(* PRIORITY 08 *)
nPriority := 8;
IF in.bR20_RC_Temperature			THEN
	out.nR20_RCTemperature			:= -1;
	fbTxBuffer[nPriority](
		IN							:= F_DIOC_20_MESSAGE_OUT(nRegister := DIOC_R01_REGISTER_REQUEST, nValue := RC_R20_RC_TEMPERATURE),
		RD							:= bTxBuffer_Read,			(* Not functional *)
		WD							:= in.bR20_RC_Temperature,
		fifo						:= ADR(TxBuffer[nPriority, 0]));
END_IF
IF in.bR21_Read_PS_AC_Voltage		THEN
	out.nR21_PsAcVoltageLevel		:= -1;
	fbTxBuffer[nPriority](
		IN							:= F_DIOC_20_MESSAGE_OUT(nRegister := DIOC_R01_REGISTER_REQUEST, nValue := RC_R21_PS_AC_VOLTAGE_LEVEL),
		RD							:= bTxBuffer_Read,			(* Not functional *)
		WD							:= in.bR21_Read_PS_AC_Voltage,
		fifo						:= ADR(TxBuffer[nPriority, 0]));
END_IF
IF in.bR22_Status_Dip_Switches		THEN
	out.sR22_Dipswitch				:= '';
	fbTxBuffer[nPriority](
		IN							:= F_DIOC_20_MESSAGE_OUT(nRegister := DIOC_R01_REGISTER_REQUEST, nValue := RC_R22_STATUS_BITS_DIPSWITCHES),
		RD							:= bTxBuffer_Read,			(* Not functional *)
		WD							:= in.bR22_Status_Dip_Switches,
		fifo						:= ADR(TxBuffer[nPriority, 0]));
END_IF
IF in.bR27_Heating_T				THEN
	out.nR27_HeatingTempHvacWater	:= -1;
	fbTxBuffer[nPriority](
		IN							:= F_DIOC_20_MESSAGE_OUT(nRegister := DIOC_R01_REGISTER_REQUEST, nValue := RC_R27_HEATING_12_13_TEMP_HVAC_WATER),
		RD							:= bTxBuffer_Read,			(* Not functional *)
		WD							:= in.bR27_Heating_T,
		fifo						:= ADR(TxBuffer[nPriority, 0]));
END_IF
IF in.bR34_Cooling_T				THEN
	out.nR34_CoolingTempIceWater	:= -1;
	fbTxBuffer[nPriority](
		IN							:= F_DIOC_20_MESSAGE_OUT(nRegister := DIOC_R01_REGISTER_REQUEST, nValue := RC_R34_COOLING_25_26_TEMP_ICE_WATER),
		RD							:= bTxBuffer_Read,			(* Not functional *)
		WD							:= in.bR34_Cooling_T,
		fifo						:= ADR(TxBuffer[nPriority, 0]));
END_IF
IF in.bR40_Pulsion_FB				THEN
	out.nR40_Pulsion_FB				:= -1;
	fbTxBuffer[nPriority](
		IN							:= F_DIOC_20_MESSAGE_OUT(nRegister := DIOC_R01_REGISTER_REQUEST, nValue := RC_R40_PULSION_17_POSITION_FEEDBACK),
		RD							:= bTxBuffer_Read,			(* Not functional *)
		WD							:= in.bR40_Pulsion_FB,
		fifo						:= ADR(TxBuffer[nPriority, 0]));
END_IF
IF in.bR42_Pulsion_T				THEN
	out.nR42_PulsionAirTemperature	:= -1;
	fbTxBuffer[nPriority](
		IN							:= F_DIOC_20_MESSAGE_OUT(nRegister := DIOC_R01_REGISTER_REQUEST, nValue := RC_R42_PULSION_18_AIR_TEMPERATURE),
		RD							:= bTxBuffer_Read,			(* Not functional *)
		WD							:= in.bR42_Pulsion_T,
		fifo						:= ADR(TxBuffer[nPriority, 0]));
END_IF
IF in.bR46_Extraction_FB			THEN
	out.nR46_Extraction_FB			:= -1;
	fbTxBuffer[nPriority](
		IN							:= F_DIOC_20_MESSAGE_OUT(nRegister := DIOC_R01_REGISTER_REQUEST, nValue := RC_R46_EXTRACTION_30_POSITION_FEEDBACK),
		RD							:= bTxBuffer_Read,			(* Not functional *)
		WD							:= in.bR46_Extraction_FB,
		fifo						:= ADR(TxBuffer[nPriority, 0]));
END_IF
IF in.bR49_Extraction_T				THEN
	out.nR49_ExtractionAirTemperature	:= -1;
	fbTxBuffer[nPriority](
		IN							:= F_DIOC_20_MESSAGE_OUT(nRegister := DIOC_R01_REGISTER_REQUEST, nValue := RC_R49_EXTRACTION_31_AIR_TEMPERATURE),
		RD							:= bTxBuffer_Read,			(* Not functional *)
		WD							:= in.bR49_Extraction_T,
		fifo						:= ADR(TxBuffer[nPriority, 0]));
END_IF
END_ACTION

ACTION Startup:
;
END_ACTION

END_FUNCTION_BLOCK

// POUs/DIOC/RC/_Internal/FB_RC_COMM
FUNCTION_BLOCK FB_RC_COMM
VAR_INPUT
	in									: ST_RC_IN;
	iPowerCycleGroup					: INT;
END_VAR
VAR_OUTPUT
	out									: ST_RC_OUT;
	nError								: E_RC_ERROR;
END_VAR
VAR CONSTANT
	TYPE_ID								: DWORD		:= 2;		(* Device identifier *)
	DEVICE_CHARGE_TIME					: TIME 		:= T#2s;	(* Optional charge time *)
	SYNC_MESSAGE_REPEAT					: TIME 		:= T#5s;	(* Sync message repeat at startup *)
	DIOC_LENGTH							: INT 		:= 21;		(* Dioc protocol length *)
	SYNC_MESSAGE						: DWORD		:= 2#0000_0000_000_1_1010_1010_1010_1111111_0;		(* Sync request = request type id *)
	SYNC_MESSAGE_HIGH					: DWORD		:= 2#0000_0000_000_1_0101_0101_0101_0101010_0;		(* Sync request = request type id *)
END_VAR
VAR
(* TC3 attribute, will be ignored by TC2 *)
{attribute 'hide_all_locals'}
(* TC2 attribute, will be ignored by TC3 *)
{library private}
	(*Startup list *)
	bStartup							: BOOL 		:= TRUE;
	bRestarted							: BOOL;					(* Device hardware restart detected by dioc *)

	(* Buffer communication *)
	Dioc_Register_IN					: ST_DIOC_REGISTER;		(* Message retrieved from buffer *)
	bRxBuffer_Read						: BOOL;
	bRxBuffer_Write						: BOOL;

	(* Fifo Buffers *)
	RxBuffer							: ARRAY[0..DIOC_RXTX_BUFFERSIZE] OF A_DIOC_MESSAGE;	(* 1 message queue *)
	TxBuffer							: ARRAY[0..DIOC_MAXPRIORITY, 0..DIOC_RXTX_BUFFERSIZE] OF A_DIOC_MESSAGE;	(* 1 message queue / priority, HIGHEST: 0 = internal priority *)

	(* Fifo Buffer handlers *)
	fbRxBuffer							: FB_DIOC_FIFO;									(* 1 message queue *)
	fbTxBuffer							: ARRAY[0..DIOC_MAXPRIORITY] OF FB_DIOC_FIFO;	(* 1 message queue / priority *)

	(* Dioc base communication layer *)
	fbDioc								: FB_DIOC;
	(* Device general register handling *)
	fbDioc_Gen							: FB_DIOC_GEN;
	(* Device specific register handling *)
	fbDioc_RC							: FB_DIOC_RC;

	i									: INT;
END_VAR

(*
	startup *)
IF bStartup THEN Startup(); END_IF
fbDioc.iPowerCycleGroup := iPowerCycleGroup;
(*
	Buffer status feedback, must be set BEFORE fb calls 
bRxBufferFull				:= fbDioc.bRxBufferFull;
bRxBufferEmpty				:= fbDioc.bRxBufferEmpty;
bTxBufferFull				:= fbDioc.bTxBufferFull;
bTxBufferEmpty				:= fbDioc.bTxBufferEmpty;*)

(*
	Get next message from message queue *)
bRxBuffer_Read				:= NOT fbDioc.out.bRxBufferEmpty;
fbRxBuffer(
	RD						:= bRxBuffer_Read,
	WD						:= bRxBuffer_Write,				(* Not functional *)
	fifo					:= ADR(RxBuffer));
Dioc_Register_IN := F_DIOC_20_MESSAGE_IN(fbRxBuffer.OUT);

(* Device Dioc base register handling and startup parameter loading *)
fbDioc_Gen(
	in						:= in.DIOC_Gen,
	in_Dioc_Status			:= fbDioc.Out,
	TYPE_ID					:= TYPE_ID,
	Dioc_Register_IN		:= Dioc_Register_IN,
	RxBuffer				:= RxBuffer,
	TxBuffer				:= TxBuffer,
	fbRxBuffer				:= fbRxBuffer,
	fbTxBuffer				:= fbTxBuffer,
	arrstStartupParameter	:= in.DIOC_RC.arrstStartupParameter,
	bRestarted				:= bRestarted,
	out						=> out.DIOC_Gen,
	nError					=>
	);
in.DIOC_Gen 				:= fbDioc_Gen.in;				(* Copy possibly changed inputs back to upper level *)

(* Device specific register handling *)
fbDioc_RC(
	in						:= in.DIOC_RC,
	in_Dioc_Status			:= fbDioc.Out,
	in_Dioc_Gen_Status		:= fbDioc_Gen.Out,
	Dioc_Register_IN		:= Dioc_Register_IN,
	RxBuffer				:= RxBuffer,
	TxBuffer				:= TxBuffer,
	fbRxBuffer				:= fbRxBuffer,
	fbTxBuffer				:= fbTxBuffer,
	bRestarted				:= bRestarted,
	out						=> out.DIOC_RC,
	nError					=>
	);
in.DIOC_RC					:= fbDioc_RC.in;				(* Copy possibly changed inputs back to upper level *)

(*
	Dioc communication layer *)
fbDioc.in.bEnable			:= in.bEnable;	(* Debug *)
fbDioc(
	DEVICE_CHARGE_TIME		:= DEVICE_CHARGE_TIME,
	DIOC_LENGTH				:= DIOC_LENGTH,
	RxBuffer				:= RxBuffer,
	TxBuffer				:= TxBuffer,
	fbRxBuffer				:= fbRxBuffer,
	fbTxBuffer				:= fbTxBuffer,
	Out						=>
	);

(*
	First loop finished *)
bStartup 					:= FALSE;

ACTION Startup:
(*
	Startup parameters *) 

(* Reset parameters
FOR i := 1 TO DIOC_NOOFSTARTUPPARAMETERS DO
	arrstStartupParameter[i].nRegister		:= 255;	(* Set to invalid *)
	arrstStartupParameter[i].nValue			:= 0;
END_FOR*)

(* Test Set parameters, switch relays
arrstStartupParameter[1].nRegister			:= 25;
arrstStartupParameter[1].nValue				:= 3;
arrstStartupParameter[2].nRegister			:= 32;
arrstStartupParameter[2].nValue				:= 3;
arrstStartupParameter[3].nRegister			:= 52;
arrstStartupParameter[3].nValue				:= 1;
arrstStartupParameter[4].nRegister			:= 25;
arrstStartupParameter[4].nValue				:= 1;
arrstStartupParameter[5].nRegister			:= 32;
arrstStartupParameter[5].nValue				:= 1;
arrstStartupParameter[6].nRegister			:= 52;
arrstStartupParameter[6].nValue				:= 2;
arrstStartupParameter[7].nRegister			:= 25;
arrstStartupParameter[7].nValue				:= 0;
arrstStartupParameter[8].nRegister			:= 32;
arrstStartupParameter[8].nValue				:= 0;
arrstStartupParameter[9].nRegister			:= 52;
arrstStartupParameter[9].nValue				:= 0;  *)


;
END_ACTION

END_FUNCTION_BLOCK

// POUs/DIOC/RC/FB_RC
FUNCTION_BLOCK FB_RC
VAR_INPUT

(*Enable bit*)
	bEn:BOOL:=TRUE; (*enable bit*)

(*input booleans*)
	bEnableFan : BOOL; (*enable fan bit (relay pin 41-42)*)

	bHeating_3P_plus :BOOL; (*Heating plus signal (output pin 7)*)
	bHeating_3P_min :BOOL; (*Heating min signal (output pin 8)*)

	bCooling_3P_plus :BOOL; (*Cooling plus signal (output pin 20)*)
	bCooling_3P_min :BOOL; (*Cooling min signal (output pin 21)*)

	bFireDamper_OPN: BOOL; (*open signal fire damper (output pin 33)*)
	bFireDamper_CLS: BOOL; (*close signal fire damper (output pin 34)*)

	bRelais_45 :BOOL; (*relay pin 45 (DO3)*)
	bRelais_46 :BOOL; (*relay pin 46 (DO2)*)
	bRelais_47 :BOOL; (*relay pin 47 (DO1)*)

(* retrieval times of all sensors*)
	iIntervalACVoltage: UDINT := 19; (*retrieval time ac voltage (in seconds)*)
	iIntervalTempHeatingWater: UDINT := 11; (*retrieval time temperature heating water (in seconds)*)
	iIntervalTempICEWater: UDINT := 9; (*retrieval time temperature ice water (in seconds)*)
	iInterval_FB_Pulsion: UDINT := 7; (*retrieval time feedback pulsion (in seconds)*)
	iIntervalTempAirPulsion: UDINT := 13; (*retrieval time temperature pulsion air (in seconds)*)
	iInterval_FB_Extraction: UDINT := 17; (*retrieval time feedback extraction (in seconds)*)
	iIntervalTempAirExtraction: UDINT := 19; (*retrieval time temperature extraction (in seconds)*)
	iIntervalDipswitches: UDINT := 17; (*retrieval time dipswitches (in seconds)*)
	iIntervalFBFiredamper: UDINT := 19; (*retrieval time feedback firedamper (in seconds)*)
	iIntervalFanFaultStatus: UDINT := 23; (*retrieval time fan fault (in seconds)*)

(* interval send times of Setpoints *)
	iSendIntervalSpHeating: INT  := 9; (*send interval time for the heating set point in seconds*)
	iSendIntervalSpCooling: INT  := 11; (*send interval time for the cooling set point in seconds*)
	iSendIntervalSpPulsion: INT  := 12; (*send interval time for the pulsion set point in seconds*)
	iSendIntervalSpExtraction: INT  := 13; (*send interval time for the extraction set point in seconds*)
	iSendIntervalSpFan: INT  := 15; (*send interval time for the fan set point in seconds*)

(* Force send setpoints *)
	bForceSendSpHeating 	: BOOL := FALSE; (*Set this to true to send the heating set point immediatly*)
	bForceSendSpCooling 	: BOOL := FALSE; (*Set this to true to send the cooling set point immediatly*)
	bForceSendSpPulsion 	: BOOL := FALSE; (*Set this to true to send the pulsion set point immediatly*)
	bForceSendSpExtraction 	: BOOL := FALSE; (*Set this to true to send the extraction set point immediatly*)
	bForceSendSpFan 		: BOOL := FALSE; (*Set this to true to send the fan set point immediatly*)

(* RC setpoints*)
	iSpHeating : INT; (*heating setpoint in %*)
	iSpCooling : INT; (*cooling setpoint in %*)
	iSpPulsion : INT; (*pulsion setpoint in %*)
	iSpExtraction : INT; (*extraction setpoint in %*)
	iSpFan : INT; (*fan setpoint in %*)

(* bool for the reset of the RC*)
	bReset:BOOL := TRUE; (*if true: resets the Room Controller*)

END_VAR
VAR_INPUT PERSISTENT

(* comment for every connection is visible on the VISU*)
	arr_sConnectionComments	: ARRAY [1..41] OF STRING(8) :=[
		'comment','comment','comment','comment','comment','comment','comment','comment','comment','comment',
		'comment','comment','comment','comment','comment','comment','comment','comment','comment','comment',
		'comment','comment','comment','comment','comment','comment','comment','comment','comment','comment',
		'comment','comment','comment','comment','comment','comment','comment','comment','comment','comment',
		'comment']; (*comments for every connection that is visible on the visualisation*)

END_VAR
VAR_OUTPUT
(*FireDamper Feedback*)
	qbFiredamperFB_OPN : BOOL; (*feedback firedamper open (input pin 37)*)
	qbFiredamperFB_CLS : BOOL; (*feedback firedamper closed (input pin 36)*)
	qbFanFault : BOOL; (*fan fault (input pin 43)*)

(* dipswitches*)
	qarr_bDipSwitches : ARRAY[1..12] OF BOOL; (*status dipswitches*)

(*measurements *)
	qfACVoltageLevel: REAL; (*measured ac voltage*)
	qfTempHeatingWater : REAL; (*temperature heating water in °C (PT1000 pin 12-13)*)
	qfTempIceWater : REAL; (*temperature ice water in °C (PT 1000 pin 25-26)*)
	qfPulsionFB : REAL; (*pulsion vav feedback in % (pin 17)*)
	qfTempAirPulsion : REAL; (*temperature pulsion in °C (PT1000 pin 18-19)*)
	qfExtractionFB : REAL; (*extraction vav feedback in % (pin 30)*)
	qfTempAirExtraction : REAL; (*temperature extraction in °C (PT1000 pin 31-32)*)

(*Analyse data*)
	qdtVersionHw: DATE;(*Hardware version of the dioc device*)
	qdtVersionSw: DATE;(*software version of the dioc device*)
	qdtVersionReg: DATE;(*register version of the dioc device*)
	qsUniqueId: STRING;(*Unique id the dioc device*)
	qrVoltageLevelA: REAL;(*Voltage level on the DIOC-A line*)
	qrVoltageLevelB: REAL;(*Voltage level on the DIOC-B line*)
	qbDeviceActive: BOOL;(*True if the device is active*)
END_VAR
VAR
(* TC3 attribute, will be ignored by TC2 *)
{attribute 'hide_all_locals'}
(* TC2 attribute, will be ignored by TC3 *)
{library private}

(*Force setpoint triggers*)
	_RtrigForceSendSpHeating: R_TRIG;
	_RtrigForceSendSpCooling: R_TRIG;
	_RtrigForceSendSpPulsion: R_TRIG;
	_RtrigForceSendSpExtraction: R_TRIG;
	_RtrigForceSendSpFan: R_TRIG;

(*SP Send Timers*)
	_tonSendIntervalSpHeating: TON;
	_tonSendIntervalSpCooling: TON;
	_tonSendIntervalSpPulsion: TON;
	_tonSendIntervalSpExtraction: TON;
	_tonSendIntervalSpFan: TON;

(* reset variabelen *)
	_iReset_Counter:INT;

(* startup variabelen *)
	_RtrigCalibration:R_TRIG;
	_FtrigCalibration:F_TRIG;
	_iLostCalibration:INT;
	_iStateInit:INT;
	_iStateInit_Counter:INT;
	_iStartupListNumber: INT := 1;
	_bFirstCycle: BOOL := TRUE;
	_iLoadbalance : INT;

(* visualisatie variabelen*)
	_iVis: INT;
	_bSelected : BOOL;
	_bAnalyse	:BOOL;
	_bPrevVisu : BOOL;
	_bNextVisu :BOOL;
	_RtrigAnalyse :R_TRIG;
	_RtrigSim :R_TRIG;
	_bSim : BOOL;
	_bComments : BOOL;

	_iSpHeatingSim : INT;
	_iSpCoolingSim : INT;
	_iSpPulsionSim : INT;
	_iSpExtractionSim : INT;
	_iSpFanSim : INT;

	_bEnableFanSim : BOOL;
	_bHeating_3P_plusSim :BOOL;
	_bHeating_3P_minSim :BOOL;
	_bCooling_3P_plusSim :BOOL;
	_bCooling_3P_minSim :BOOL;
	_bFireDamper_OPNSim: BOOL;
	_bFireDamper_CLSSim: BOOL;
	_bRelais_45Sim : BOOL;
	_bRelais_46Sim : BOOL;
	_bRelais_47Sim : BOOL;

(*start*)
	_bInit : BOOL := FALSE;

(*functionblock for communication with RC *)
	FB_DIOC_COMM : FB_RC_COMM;

END_VAR

(*Wait 0.5s to start the next DIOC device, charging too many DIOC devices at once will give too much current*)
IF NOT _bInit THEN
    DIOC_tonLastStart(IN:=TRUE , PT:= T#500ms);
    IF  NOT DIOC_tonLastStart.Q THEN
    	RETURN;
    END_IF
    DIOC_tonLastStart(IN:=FALSE , PT:= T#500ms); (*resets the timer*)
    _bInit := TRUE;
END_IF

(* falling and rising edge RC calibration*)
_RtrigCalibration(CLK:= FB_DIOC_COMM.out.DIOC_Gen.bDeviceActive, Q=> );
_FtrigCalibration(CLK:= FB_DIOC_COMM.out.DIOC_Gen.bDeviceActive, Q=> );

(* enable reset the device when calibration is lost for 30 cycles. *)
IF _FtrigCalibration.Q THEN
	_iLostCalibration := 1;
END_IF

IF _iLostCalibration = 30 THEN
	bReset := TRUE;
END_IF

IF _iLostCalibration < 30 AND _iLostCalibration > 0 AND NOT FB_DIOC_COMM.out.DIOC_Gen.bDeviceActive THEN
	_iLostCalibration := _iLostCalibration + 1;
ELSE
	_iLostCalibration := 0;
END_IF

(* reset the device when breset is high, cut off power to device for 1000 cycles to make sure the device has lost all power*)
IF breset OR DIOC_bRestart OR NOT bEn THEN
	_iReset_Counter := 0;
	FB_DIOC_COMM.in.bEnable := FALSE;
	breset := FALSE;
END_IF

IF _iReset_Counter < 1000 THEN
	IF _iReset_Counter = 999 THEN
	    _bInit := FALSE;
	END_IF
	_iReset_Counter := _iReset_Counter +1;
	_iStateInit := 0;
ELSE
	FB_DIOC_COMM.in.bEnable := bEn;
END_IF

(* send startuplist, send all values that need to be sent at startup + set automatic response types of certain measurements,
with synchronisations added in between the messages to not disrupt the flow of the startparameters *)

IF _bFirstCycle THEN
	StartupList();
END_IF

(* request all static info when the device has been active for some time *)
stateinit();

_RtrigSim(CLK:= _bSim, Q=> );
IF _RtrigSim.q THEN
	(* limit analog values from 0% to 100% *)
	iSpHeating := LIMIT(0,iSpHeating,100);
	iSpCooling := LIMIT(0,iSpCooling,100);
	iSpPulsion := LIMIT(0,iSpPulsion,100);
	iSpExtraction := LIMIT(0,iSpExtraction,100);
	iSpFan := LIMIT(0,iSpFan,100);

	_iSpHeatingSim  := iSpHeating;
	_iSpCoolingSim  := iSpCooling;
	_iSpPulsionSim  := iSpPulsion;
	_iSpExtractionSim  := iSpExtraction;
	_iSpFanSim  := iSpFan;

	_bEnableFanSim := bEnableFan;
	_bHeating_3P_plusSim := bHeating_3P_plus;
	_bHeating_3P_minSim := bHeating_3P_min;
	_bCooling_3P_plusSim := bCooling_3P_plus;
	_bCooling_3P_minSim := bCooling_3P_min;
	_bFireDamper_OPNSim:= bFireDamper_OPN;
	_bFireDamper_CLSSim:= bFireDamper_CLS;
END_IF

(*Forward setpoints*)
_RtrigForceSendSpHeating(CLK:= bForceSendSpHeating);
bForceSendSpHeating := FALSE;
_tonSendIntervalSpHeating(IN:= NOT _tonSendIntervalSpHeating.q, PT:= UDINT_TO_TIME(INT_TO_UDINT(iSendIntervalSpHeating * 1000)));
IF _tonSendIntervalSpHeating.Q OR _RtrigForceSendSpHeating.Q THEN
	(* limit analog values from 0% to 100% *)
	iSpHeating := LIMIT(0,iSpHeating,100);
	FB_DIOC_COMM.in.DIOC_RC.nR26_Heating_SP := INT_TO_UINT(TRUNC_INT(INT_TO_REAL( SEL(_bSim, iSpHeating, _iSpHeatingSim)) / 100* 4090));
	FB_DIOC_COMM.in.DIOC_RC.bR26_Heating_SP := TRUE;
END_IF;

_RtrigForceSendSpCooling(CLK:= bForceSendSpCooling);
bForceSendSpCooling := FALSE;
_tonSendIntervalSpCooling(IN:= NOT _tonSendIntervalSpCooling.q, PT:= UDINT_TO_TIME(INT_TO_UDINT(iSendIntervalSpCooling * 1000)));
IF _tonSendIntervalSpCooling.Q OR _RtrigForceSendSpCooling.Q  THEN
	(* limit analog values from 0% to 100% *)
	iSpCooling := LIMIT(0,iSpCooling,100);
	FB_DIOC_COMM.in.DIOC_RC.nR33_Cooling_SP := INT_TO_UINT(TRUNC_INT(INT_TO_REAL( SEL(_bSim, iSpCooling, _iSpCoolingSim)) / 100* 4090));
	FB_DIOC_COMM.in.DIOC_RC.bR33_Cooling_SP := TRUE;
END_IF;

_RtrigForceSendSpPulsion(CLK:= bForceSendSpPulsion);
bForceSendSpPulsion := FALSE;
_tonSendIntervalSpPulsion(IN:= NOT _tonSendIntervalSpPulsion.q, PT:= UDINT_TO_TIME(INT_TO_UDINT(iSendIntervalSpPulsion * 1000)));
IF _tonSendIntervalSpPulsion.Q OR _RtrigForceSendSpPulsion.Q   THEN
	(* limit analog values from 0% to 100% *)
	iSpPulsion := LIMIT(0,iSpPulsion,100);
	FB_DIOC_COMM.in.DIOC_RC.nR39_Pulsion_SP := INT_TO_UINT(TRUNC_INT(INT_TO_REAL( SEL(_bSim, iSpPulsion, _iSpPulsionSim)) / 100* 4090));
	FB_DIOC_COMM.in.DIOC_RC.bR39_Pulsion_SP := TRUE;
END_IF;

_RtrigForceSendSpExtraction(CLK:= bForceSendSpExtraction);
bForceSendSpExtraction := FALSE;
_tonSendIntervalSpExtraction(IN:= NOT _tonSendIntervalSpExtraction.q, PT:= UDINT_TO_TIME(INT_TO_UDINT(iSendIntervalSpExtraction * 1000)));
IF _tonSendIntervalSpExtraction.Q OR _RtrigForceSendSpExtraction.Q   THEN
	(* limit analog values from 0% to 100% *)
	iSpExtraction := LIMIT(0,iSpExtraction,100);
	FB_DIOC_COMM.in.DIOC_RC.nR45_Extraction_SP := INT_TO_UINT(TRUNC_INT(INT_TO_REAL( SEL(_bSim, iSpExtraction, _iSpExtractionSim)) / 100* 4090));
	FB_DIOC_COMM.in.DIOC_RC.bR45_Extraction_SP := TRUE;
END_IF;

_RtrigForceSendSpFan(CLK:= bForceSendSpFan);
bForceSendSpFan := FALSE;
_tonSendIntervalSpFan(IN:= NOT _tonSendIntervalSpFan.q, PT:= UDINT_TO_TIME(INT_TO_UDINT(iSendIntervalSpFan * 1000)));
IF _tonSendIntervalSpFan.Q  OR _RtrigForceSendSpFan.Q  THEN
	(* limit analog values from 0% to 100% *)
	iSpFan := LIMIT(0,iSpFan,100);
	FB_DIOC_COMM.in.DIOC_RC.nR56_Fan_SP := INT_TO_UINT(TRUNC_INT(INT_TO_REAL( SEL(_bSim, iSpFan, _iSpFanSim)) /100* 4090));
	FB_DIOC_COMM.in.DIOC_RC.bR56_Fan_SP := TRUE;
END_IF;

(* call communication block *)
FB_DIOC_COMM(in:= , out=> , nError=> );

(*Inputs*)
qarr_bDipSwitches[1] := FB_DIOC_COMM.out.DIOC_RC.bR22_Dipswitch_S01;
qarr_bDipSwitches[2] := FB_DIOC_COMM.out.DIOC_RC.bR22_Dipswitch_S02;
qarr_bDipSwitches[3] := FB_DIOC_COMM.out.DIOC_RC.bR22_Dipswitch_S03;
qarr_bDipSwitches[4] := FB_DIOC_COMM.out.DIOC_RC.bR22_Dipswitch_S04;
qarr_bDipSwitches[5] := FB_DIOC_COMM.out.DIOC_RC.bR22_Dipswitch_S05;
qarr_bDipSwitches[6] := FB_DIOC_COMM.out.DIOC_RC.bR22_Dipswitch_S06;
qarr_bDipSwitches[7] := FB_DIOC_COMM.out.DIOC_RC.bR22_Dipswitch_S07;
qarr_bDipSwitches[8] := FB_DIOC_COMM.out.DIOC_RC.bR22_Dipswitch_S08;
qarr_bDipSwitches[9] := FB_DIOC_COMM.out.DIOC_RC.bR22_Dipswitch_S09;
qarr_bDipSwitches[10] := FB_DIOC_COMM.out.DIOC_RC.bR22_Dipswitch_S10;
qarr_bDipSwitches[11] := FB_DIOC_COMM.out.DIOC_RC.bR22_Dipswitch_S11;
qarr_bDipSwitches[12] := FB_DIOC_COMM.out.DIOC_RC.bR22_Dipswitch_S12;

qbFiredamperFB_OPN := FB_DIOC_COMM.out.DIOC_RC.bR53_FireDamperFB_OPN;
qbFiredamperFB_CLS := FB_DIOC_COMM.out.DIOC_RC.bR53_FireDamperFB_CLS;
qbFanFault := FB_DIOC_COMM.out.DIOC_RC.bR58_FanFaultStatus;

(*Measurements *)
qfACVoltageLevel:=FB_DIOC_COMM.out.DIOC_RC.nR21_PsAcVoltageLevel;
qfTempHeatingWater:=FB_DIOC_COMM.out.DIOC_RC.nR27_HeatingTempHvacWater;
qfTempIceWater:=FB_DIOC_COMM.out.DIOC_RC.nR34_CoolingTempIceWater;
qfPulsionFB:=FB_DIOC_COMM.out.DIOC_RC.nR40_Pulsion_FB;
qfTempAirPulsion:=FB_DIOC_COMM.out.DIOC_RC.nR42_PulsionAirTemperature;
qfExtractionFB:=FB_DIOC_COMM.out.DIOC_RC.nR46_Extraction_FB;
qfTempAirExtraction:=FB_DIOC_COMM.out.DIOC_RC.nR49_ExtractionAirTemperature;

(*Outputs*)
FB_DIOC_COMM.in.DIOC_RC.bR25_Heating_7_8_3p_min := SEL(_bSim, bHeating_3P_min, _bHeating_3P_minSim);
FB_DIOC_COMM.in.DIOC_RC.bR25_Heating_7_8_3p_plus_pwm := SEL(_bSim, bHeating_3P_plus, _bHeating_3P_plusSim);

FB_DIOC_COMM.in.DIOC_RC.bR32_Cooling_20_21_3p_min := SEL(_bSim, bCooling_3P_min, _bCooling_3P_minSim);
FB_DIOC_COMM.in.DIOC_RC.bR32_Cooling_20_21_3p_plus_pwm := SEL(_bSim, bCooling_3P_plus, _bCooling_3P_plusSim);

FB_DIOC_COMM.in.DIOC_RC.bR52_FireDamperCOM_NC := SEL(_bSim, bFireDamper_CLS, _bFireDamper_CLSSim);
FB_DIOC_COMM.in.DIOC_RC.bR52_FireDamperCOM_NO := SEL(_bSim, bFireDamper_OPN, _bFireDamper_OPNSim);

FB_DIOC_COMM.in.DIOC_RC.bR57_Fan_Enable := SEL(_bSim, bEnableFan, _bEnableFanSim);

FB_DIOC_COMM.in.DIOC_RC.bR61_do_45 := SEL(_bSim, bRelais_45, _bRelais_45Sim);
FB_DIOC_COMM.in.DIOC_RC.bR61_do_46 := SEL(_bSim, bRelais_46, _bRelais_46Sim);
FB_DIOC_COMM.in.DIOC_RC.bR61_do_47 := SEL(_bSim, bRelais_47, _bRelais_47Sim);


(*loadbalance, only do these tasks every 47 cycles to save time *)
_iLoadbalance := _iLoadbalance + 1;
IF _iLoadbalance > 47 THEN
	_iLoadbalance := 0;

	(*save static info*)
	qdtVersionHw:=FB_DIOC_COMM.out.DIOC_Gen.dtR04_VersionHW;
	qdtVersionSw:=FB_DIOC_COMM.out.DIOC_Gen.dtR05_VersionSW;
	qdtVersionReg:=FB_DIOC_COMM.out.DIOC_Gen.dtR06_VersionREG;
	qsUniqueId:=FB_DIOC_COMM.out.DIOC_Gen.sR07_UniqueID;
	
	qrVoltageLevelA:=FB_DIOC_COMM.out.DIOC_Gen.nR09_DiocVoltageA;
	qrVoltageLevelB:=FB_DIOC_COMM.out.DIOC_Gen.nR10_DiocVoltageB;

	qbDeviceActive:=FB_DIOC_COMM.out.DIOC_Gen.bDeviceActive;
END_IF;

(* Visualisation *)
(*
_RtrigAnalyse(CLK:= _bAnalyse, Q=> );
IF _RtrigAnalyse.q  AND (CurrentVisu <> DIOC_DEBUGSCHERM) AND DIOC_Debug THEN
	DIOC_DebugLinkPrevScreen:=CurrentVisu;
	CurrentVisu := DIOC_DEBUGSCHERM;
END_IF
IF _bAnalyse AND DIOC_Debug THEN
	DIOC_pDebugged_RC := ADRINST();
	_bAnalyse := FALSE;
END_IF*)

IF _bSelected = FALSE THEN
	_bSim := FALSE;
	_iVis := 0;
END_IF;

IF _bNextVisu THEN
	_iVis := _iVis + 1;
	_bNextVisu := FALSE;
END_IF

IF _bPrevVisu THEN
	_iVis := _iVis - 1;
	_bPrevVisu := FALSE;
END_IF

IF _iVis > 0 THEN
	_iVis := 0;
END_IF;

IF _iVis < 0 THEN
	_iVis := 0;
END_IF;

_bFirstCycle := FALSE;

ACTION StartupList:
_iStartupListNumber := 1;
(*change transmit offset*)
FB_DIOC_COMM.in.DIOC_RC.arrstStartupParameter[_iStartupListNumber].nRegister:=DIOC_R84_TRANSMIT_DELAY;
FB_DIOC_COMM.in.DIOC_RC.arrstStartupParameter[_iStartupListNumber].nValue:=30;

_iStartupListNumber := _iStartupListNumber +1;
FB_DIOC_COMM.in.DIOC_RC.arrstStartupParameter[_iStartupListNumber].nRegister:=DIOC_R02_REGISTER_INTERVAL;
FB_DIOC_COMM.in.DIOC_RC.arrstStartupParameter[_iStartupListNumber].nValue:=19;

_iStartupListNumber := _iStartupListNumber +1;
FB_DIOC_COMM.in.DIOC_RC.arrstStartupParameter[_iStartupListNumber].nRegister:=DIOC_R01_REGISTER_REQUEST;
FB_DIOC_COMM.in.DIOC_RC.arrstStartupParameter[_iStartupListNumber].nValue:=INT_TO_DWORD(DIOC_R84_TRANSMIT_DELAY);

(*device enabled*)
FB_DIOC_COMM.in.DIOC_RC.arrstStartupParameter[_iStartupListNumber].nRegister:=DIOC_R02_REGISTER_INTERVAL;
FB_DIOC_COMM.in.DIOC_RC.arrstStartupParameter[_iStartupListNumber].nValue:=15;

_iStartupListNumber := _iStartupListNumber +1;
FB_DIOC_COMM.in.DIOC_RC.arrstStartupParameter[_iStartupListNumber].nRegister:=DIOC_R01_REGISTER_REQUEST;
FB_DIOC_COMM.in.DIOC_RC.arrstStartupParameter[_iStartupListNumber].nValue:=INT_TO_DWORD(DIOC_R11_DEVICE_ENABLE);

(*voltage level A*)
_iStartupListNumber := _iStartupListNumber +1;
FB_DIOC_COMM.in.DIOC_RC.arrstStartupParameter[_iStartupListNumber].nRegister:=DIOC_R02_REGISTER_INTERVAL;
FB_DIOC_COMM.in.DIOC_RC.arrstStartupParameter[_iStartupListNumber].nValue:=59;

_iStartupListNumber := _iStartupListNumber +1;
FB_DIOC_COMM.in.DIOC_RC.arrstStartupParameter[_iStartupListNumber].nRegister:=DIOC_R01_REGISTER_REQUEST;
FB_DIOC_COMM.in.DIOC_RC.arrstStartupParameter[_iStartupListNumber].nValue:=INT_TO_DWORD(DIOC_R09_VOLTAGE_LEVEL_A);

(*voltage level B*)
_iStartupListNumber := _iStartupListNumber +1;
FB_DIOC_COMM.in.DIOC_RC.arrstStartupParameter[_iStartupListNumber].nRegister:=DIOC_R02_REGISTER_INTERVAL;
FB_DIOC_COMM.in.DIOC_RC.arrstStartupParameter[_iStartupListNumber].nValue:=61;

_iStartupListNumber := _iStartupListNumber +1;
FB_DIOC_COMM.in.DIOC_RC.arrstStartupParameter[_iStartupListNumber].nRegister:=DIOC_R01_REGISTER_REQUEST;
FB_DIOC_COMM.in.DIOC_RC.arrstStartupParameter[_iStartupListNumber].nValue:=INT_TO_DWORD(DIOC_R10_VOLTAGE_LEVEL_B);

(*AC PS Voltage level*)
_iStartupListNumber := _iStartupListNumber +1;
FB_DIOC_COMM.in.DIOC_RC.arrstStartupParameter[_iStartupListNumber].nRegister:=DIOC_R02_REGISTER_INTERVAL;
FB_DIOC_COMM.in.DIOC_RC.arrstStartupParameter[_iStartupListNumber].nValue:=iIntervalACVoltage;

_iStartupListNumber := _iStartupListNumber +1;
FB_DIOC_COMM.in.DIOC_RC.arrstStartupParameter[_iStartupListNumber].nRegister:=DIOC_R01_REGISTER_REQUEST;
FB_DIOC_COMM.in.DIOC_RC.arrstStartupParameter[_iStartupListNumber].nValue:=INT_TO_DWORD(RC_R21_PS_AC_VOLTAGE_LEVEL);

(* Heating 12-13 temperature HVAC water *)
_iStartupListNumber := _iStartupListNumber +1;
FB_DIOC_COMM.in.DIOC_RC.arrstStartupParameter[_iStartupListNumber].nRegister:=DIOC_R02_REGISTER_INTERVAL;
FB_DIOC_COMM.in.DIOC_RC.arrstStartupParameter[_iStartupListNumber].nValue:=iIntervalTempHeatingWater;

_iStartupListNumber := _iStartupListNumber +1;
FB_DIOC_COMM.in.DIOC_RC.arrstStartupParameter[_iStartupListNumber].nRegister:=DIOC_R01_REGISTER_REQUEST;
FB_DIOC_COMM.in.DIOC_RC.arrstStartupParameter[_iStartupListNumber].nValue:= INT_TO_DWORD(RC_R27_HEATING_12_13_TEMP_HVAC_WATER);

(*sync*)
_iStartupListNumber := _iStartupListNumber +1;
FB_DIOC_COMM.in.DIOC_RC.arrstStartupParameter[_iStartupListNumber].nRegister:=85;
FB_DIOC_COMM.in.DIOC_RC.arrstStartupParameter[_iStartupListNumber].nValue:=2730;

(*Cooling 25-26 temperature ICE water *)
_iStartupListNumber := _iStartupListNumber +1;
FB_DIOC_COMM.in.DIOC_RC.arrstStartupParameter[_iStartupListNumber].nRegister:=DIOC_R02_REGISTER_INTERVAL;
FB_DIOC_COMM.in.DIOC_RC.arrstStartupParameter[_iStartupListNumber].nValue:=iIntervalTempICEWater;

_iStartupListNumber := _iStartupListNumber +1;
FB_DIOC_COMM.in.DIOC_RC.arrstStartupParameter[_iStartupListNumber].nRegister:=DIOC_R01_REGISTER_REQUEST;
FB_DIOC_COMM.in.DIOC_RC.arrstStartupParameter[_iStartupListNumber].nValue:=INT_TO_DWORD(RC_R34_COOLING_25_26_TEMP_ICE_WATER);

(* Pulsion_FB *)
_iStartupListNumber := _iStartupListNumber +1;
FB_DIOC_COMM.in.DIOC_RC.arrstStartupParameter[_iStartupListNumber].nRegister:=DIOC_R02_REGISTER_INTERVAL;
FB_DIOC_COMM.in.DIOC_RC.arrstStartupParameter[_iStartupListNumber].nValue:=iInterval_FB_Pulsion;

_iStartupListNumber := _iStartupListNumber +1;
FB_DIOC_COMM.in.DIOC_RC.arrstStartupParameter[_iStartupListNumber].nRegister:=DIOC_R01_REGISTER_REQUEST;
FB_DIOC_COMM.in.DIOC_RC.arrstStartupParameter[_iStartupListNumber].nValue:=INT_TO_DWORD(RC_R40_PULSION_17_POSITION_FEEDBACK);

(* Pulsion Air Temperature *)
_iStartupListNumber := _iStartupListNumber +1;
FB_DIOC_COMM.in.DIOC_RC.arrstStartupParameter[_iStartupListNumber].nRegister:=DIOC_R02_REGISTER_INTERVAL;
FB_DIOC_COMM.in.DIOC_RC.arrstStartupParameter[_iStartupListNumber].nValue:=iIntervalTempAirPulsion;

_iStartupListNumber := _iStartupListNumber +1;
FB_DIOC_COMM.in.DIOC_RC.arrstStartupParameter[_iStartupListNumber].nRegister:=DIOC_R01_REGISTER_REQUEST;
FB_DIOC_COMM.in.DIOC_RC.arrstStartupParameter[_iStartupListNumber].nValue:=INT_TO_DWORD(RC_R42_PULSION_18_AIR_TEMPERATURE);

(*sync*)
_iStartupListNumber := _iStartupListNumber +1;
FB_DIOC_COMM.in.DIOC_RC.arrstStartupParameter[_iStartupListNumber].nRegister:=85;
FB_DIOC_COMM.in.DIOC_RC.arrstStartupParameter[_iStartupListNumber].nValue:=2730;

(* Extraction_FB *)
_iStartupListNumber := _iStartupListNumber +1;
FB_DIOC_COMM.in.DIOC_RC.arrstStartupParameter[_iStartupListNumber].nRegister:=DIOC_R02_REGISTER_INTERVAL;
FB_DIOC_COMM.in.DIOC_RC.arrstStartupParameter[_iStartupListNumber].nValue:=iInterval_FB_Extraction;

_iStartupListNumber := _iStartupListNumber +1;
FB_DIOC_COMM.in.DIOC_RC.arrstStartupParameter[_iStartupListNumber].nRegister:=DIOC_R01_REGISTER_REQUEST;
FB_DIOC_COMM.in.DIOC_RC.arrstStartupParameter[_iStartupListNumber].nValue:=INT_TO_DWORD(RC_R46_EXTRACTION_30_POSITION_FEEDBACK);

(* Extraction Air Temperature *)
_iStartupListNumber := _iStartupListNumber +1;
FB_DIOC_COMM.in.DIOC_RC.arrstStartupParameter[_iStartupListNumber].nRegister:=DIOC_R02_REGISTER_INTERVAL;
FB_DIOC_COMM.in.DIOC_RC.arrstStartupParameter[_iStartupListNumber].nValue:=iIntervalTempAirExtraction;

_iStartupListNumber := _iStartupListNumber +1;
FB_DIOC_COMM.in.DIOC_RC.arrstStartupParameter[_iStartupListNumber].nRegister:=DIOC_R01_REGISTER_REQUEST;
FB_DIOC_COMM.in.DIOC_RC.arrstStartupParameter[_iStartupListNumber].nValue:=INT_TO_DWORD(RC_R49_EXTRACTION_31_AIR_TEMPERATURE);

(* Dipswitches *)
_iStartupListNumber := _iStartupListNumber +1;
FB_DIOC_COMM.in.DIOC_RC.arrstStartupParameter[_iStartupListNumber].nRegister:=DIOC_R02_REGISTER_INTERVAL;
FB_DIOC_COMM.in.DIOC_RC.arrstStartupParameter[_iStartupListNumber].nValue:=iIntervalDipswitches;

_iStartupListNumber := _iStartupListNumber +1;
FB_DIOC_COMM.in.DIOC_RC.arrstStartupParameter[_iStartupListNumber].nRegister:=DIOC_R01_REGISTER_REQUEST;
FB_DIOC_COMM.in.DIOC_RC.arrstStartupParameter[_iStartupListNumber].nValue:=INT_TO_DWORD(RC_R22_STATUS_BITS_DIPSWITCHES);

(* FB_Firedamper *)
_iStartupListNumber := _iStartupListNumber +1;
FB_DIOC_COMM.in.DIOC_RC.arrstStartupParameter[_iStartupListNumber].nRegister:=DIOC_R02_REGISTER_INTERVAL;
FB_DIOC_COMM.in.DIOC_RC.arrstStartupParameter[_iStartupListNumber].nValue:=iIntervalFBFiredamper;

_iStartupListNumber := _iStartupListNumber +1;
FB_DIOC_COMM.in.DIOC_RC.arrstStartupParameter[_iStartupListNumber].nRegister:=DIOC_R01_REGISTER_REQUEST;
FB_DIOC_COMM.in.DIOC_RC.arrstStartupParameter[_iStartupListNumber].nValue:=INT_TO_DWORD(RC_R53_FIREDAMPER_36_37_FEEDBACK);

(* fan fault status *)
_iStartupListNumber := _iStartupListNumber +1;
FB_DIOC_COMM.in.DIOC_RC.arrstStartupParameter[_iStartupListNumber].nRegister:=DIOC_R02_REGISTER_INTERVAL;
FB_DIOC_COMM.in.DIOC_RC.arrstStartupParameter[_iStartupListNumber].nValue:=iIntervalFanFaultStatus;

_iStartupListNumber := _iStartupListNumber +1;
FB_DIOC_COMM.in.DIOC_RC.arrstStartupParameter[_iStartupListNumber].nRegister:=DIOC_R01_REGISTER_REQUEST;
FB_DIOC_COMM.in.DIOC_RC.arrstStartupParameter[_iStartupListNumber].nValue:=INT_TO_DWORD(RC_R58_FAN_FAULT_STATUS);

(*sync*)
_iStartupListNumber := _iStartupListNumber +1;
FB_DIOC_COMM.in.DIOC_RC.arrstStartupParameter[_iStartupListNumber].nRegister:=85;
FB_DIOC_COMM.in.DIOC_RC.arrstStartupParameter[_iStartupListNumber].nValue:=2730;
END_ACTION

ACTION Stateinit:
(* Gradually request all static information at startup of the RC *)
CASE _iStateInit OF
	0:
		IF _RtrigCalibration.Q  THEN
		_iStateInit:=1;
		END_IF
	1:
		_iStateInit_Counter:=_iStateInit_Counter+1;
		IF _iStateInit_Counter>4000 THEN
			_iStateInit:=_iStateInit+1;
			_iStateInit_Counter:=0;
		END_IF
	2:
		FB_DIOC_COMM.in.DIOC_Gen.bR04_Request_HW_Version:=TRUE;
		_iStateInit:=_iStateInit+1;
	3:
		_iStateInit_Counter:=_iStateInit_Counter+1;
		IF FB_DIOC_COMM.out.DIOC_Gen.dtR04_VersionHW <> DWORD_TO_DATE(0) THEN
			_iStateInit:=_iStateInit+1;
			_iStateInit_Counter:=0;
		ELSE
			IF _iStateInit_Counter>1000 THEN
				FB_DIOC_COMM.in.DIOC_Gen.bR04_Request_HW_Version:=TRUE;
				_iStateInit_Counter:=0;
			END_IF
		END_IF
	4:
		FB_DIOC_COMM.in.DIOC_Gen.bR05_Request_SW_Version:=TRUE;
		_iStateInit:=_iStateInit+1;
	5:
			_iStateInit_Counter:=_iStateInit_Counter+1;
		IF FB_DIOC_COMM.out.DIOC_Gen.dtR05_VersionSW <> DWORD_TO_DATE(0) THEN
			_iStateInit:=_iStateInit+1;
			_iStateInit_Counter:=0;
		ELSE
			IF _iStateInit_Counter>1000 THEN
				FB_DIOC_COMM.in.DIOC_Gen.bR05_Request_SW_Version:=TRUE;
				_iStateInit_Counter:=0;
			END_IF
		END_IF
	6:
		FB_DIOC_COMM.in.DIOC_Gen.bR06_Request_Register_Version:=TRUE;
		_iStateInit:=_iStateInit+1;
	7:
			_iStateInit_Counter:=_iStateInit_Counter+1;
		IF FB_DIOC_COMM.out.DIOC_Gen.dtR06_VersionREG <> DWORD_TO_DATE(0) THEN
			_iStateInit:=_iStateInit+1;
			_iStateInit_Counter:=0;
		ELSE
			IF _iStateInit_Counter>1000 THEN
				FB_DIOC_COMM.in.DIOC_Gen.bR06_Request_Register_Version:=TRUE;
				_iStateInit_Counter:=0;
			END_IF
		END_IF
	8:
		FB_DIOC_COMM.in.DIOC_Gen.bR07_Request_Unique_ID:=TRUE;
		_iStateInit:=_iStateInit+1;
	9:
		_iStateInit_Counter:=_iStateInit_Counter+1;
		IF FB_DIOC_COMM.out.DIOC_Gen.sR07_UniqueID <> '' THEN
			_iStateInit:=_iStateInit+1;
			_iStateInit_Counter:=0;
		ELSE
			IF _iStateInit_Counter>800 THEN
				FB_DIOC_COMM.in.DIOC_Gen.bR07_Request_Unique_ID:=TRUE;
				_iStateInit_Counter:=0;
			END_IF
		END_IF
	10:
		_iStateInit := 0;
END_CASE
END_ACTION

END_FUNCTION_BLOCK

// POUs/DIOC/TP10/_Internal/FB_DIOC_TP10
FUNCTION_BLOCK FB_DIOC_TP10
VAR_INPUT
	(* Data handshake interface *)
	in									: ST_DIOC_TP10_IN;
	in_Dioc_Status						: ST_DIOC_OUT;			(* Feedback dioc communication block *)
	in_Dioc_Gen_Status					: ST_DIOC_GEN_OUT;		(* Feedback general registers *)
	(*bDeviceReady						: BOOL;					(* Device charged and ready *)
	bDeviceActive						: BOOL;					(* Device is active *)*)
	Dioc_Register_IN					: ST_DIOC_REGISTER;		(* Message retrieved from buffer *)
	(* Buffer statusses *)
	bRxBufferFull						: BOOL;
	bRxBufferEmpty						: BOOL;
	bTxBufferFull						: BOOL;
	bTxBufferEmpty						: BOOL;
END_VAR
VAR_OUTPUT
	(* RC feedback data *)
	out									: ST_DIOC_TP10_OUT;
	nError								: E_DIOC_TP10_ERROR;
	qbBufferFull						: BOOL;
END_VAR
VAR_IN_OUT
	(*Dioc_Register_OUT					: A_DIOC_MESSAGE;*)
	RxBuffer							: ARRAY[0..DIOC_RXTX_BUFFERSIZE] OF A_DIOC_MESSAGE;	(* 1 message queue *)
	TxBuffer							: ARRAY[0..DIOC_MAXPRIORITY, 0..DIOC_RXTX_BUFFERSIZE] OF A_DIOC_MESSAGE;	(* 1 message queue / priority, HIGHEST: 0 = internal priority *)
	(* Fifo Buffer handlers *)
	fbRxBuffer							: FB_DIOC_FIFO;									(* 1 message queue *)
	fbTxBuffer							: ARRAY[0..DIOC_MAXPRIORITY] OF FB_DIOC_FIFO;	(* 1 message queue / priority *)
	(* Restarted ? *)
	bRestarted							: BOOL;
END_VAR
VAR
(* TC3 attribute, will be ignored by TC2 *)
{attribute 'hide_all_locals'}
(* TC2 attribute, will be ignored by TC3 *)
{library private}
	(* Previous state in *)
	stDeviceDataInPrevious				: ST_DIOC_TP10_IN;

	(*
		Timer sync message *)
	tSync								: TON;

	(*
		dioc communication *)
	stDiocRegister						: ST_DIOC_REGISTER;
	stDiocMessage						: A_DIOC_MESSAGE;

	(*
		Sync message response, response is constructed at runtime, can depend on device *)
	dwSyncMessageResponse				: DWORD;

	(*
		device data IN, request to the device *)
	fpDeviceDataInNew					: R_TRIG;

	(*
		Startup list *)
	bStartup							: BOOL 		:= TRUE;

	iRefreshCycles						: INT;
	_FtrigCalibration					:F_TRIG;

	(* various *)
	i									: INT;
	byToggle							: BYTE;
	nPriority							: INT;		(* This value avoids copy paste errors, filled in by the program, see send action *)

	(* TEMP VARS *)
	nWriteRegister				 		: A_DIOC_DATA_TYPE;
	(* Buffer read / write *)
	bRxBuffer_Read						: BOOL;
	bRxBuffer_Write						: BOOL;
	bTxBuffer_Read						: BOOL;
	bTxBuffer_Write						: BOOL;

	(* Current values *)
	sR07_UniqueID						: STRING[24];				(* TEMP R7: Unique ID *)
	sR07_UniqueID_hex					: STRING[2];				(* TEMP R7: Unique ID *)

	nTemp: DINT;
	byParity							: BYTE; (*Byte to determine parity*)
	iNoButtonParity: INT;


	outRef									: ST_DIOC_TP10_OUT;
END_VAR

(* © 2016 FixSus BVBA all rights reserved *)
(* © Handles TP10 specific variables of the TP10 *)
(*	startup *)
IF bStartup THEN Startup(); END_IF

(*
	Toggle byte *)
byToggle		:= byToggle + 1;

(* handle restart *)
IF	bRestarted				THEN
	Restart();
END_IF

(*refresh sent data every 1000 cycles*)
IF iRefreshCycles < 1000 THEN
	iRefreshCycles := iRefreshCycles +1;
ELSIF in_Dioc_Gen_Status.nR10_DiocVoltageB > -1 THEN
	iRefreshCycles := 0;
END_IF;

(*on loss of calibration reset all values to 0*)
_FtrigCalibration(CLK:= in_Dioc_Gen_Status.bDeviceActive, Q=> );

IF _FtrigCalibration.Q THEN
	out.nR50_TouchButtonStatus			:= 0;
	out.bR50_TouchButton01				:= out.nR50_TouchButtonStatus.0;
	out.bR50_TouchButton02				:= out.nR50_TouchButtonStatus.1;
	out.bR50_TouchButton03				:= out.nR50_TouchButtonStatus.2;
	out.bR50_TouchButton04				:= out.nR50_TouchButtonStatus.3;
	out.bR50_TouchButton05				:= out.nR50_TouchButtonStatus.4;
	out.bR50_TouchButton06				:= out.nR50_TouchButtonStatus.5;
	out.bR50_TouchButton07				:= out.nR50_TouchButtonStatus.6;
	out.bR50_TouchButton08				:= out.nR50_TouchButtonStatus.7;
	out.bR50_TouchButton09				:= out.nR50_TouchButtonStatus.8;
	out.bR50_TouchButton10				:= out.nR50_TouchButtonStatus.9;
	out.nR21_RoomTemperature 			:= 0;
	out.nR27_VOC			 			:= 0;
	out.nR25_CO2			 			:= 0;
	out.nR23_ROOM_HUMIDITY	 			:= 0;
	out.nR35_ROOM_ILLUMINATION_LUXL_VALUE 	:= 0;
	out.nR36_ROOM_ILLUMINATION_LUXH_VALUE	:= 0;
	out.nR37_ROOM_ILLUMINATION_IRL_VALUE 	:= 0;
	out.nR38_ROOM_ILLUMINATION_IRH_VALUE 	:= 0;
END_IF;
(*
	Process new data from dioc *)
Receive();

(*
	External Dioc request processing, with priority handling *)
Send();

(*
	First loop finished *)
bStartup 					:= FALSE;

ACTION Receive:
(* !!! ONLY ACTIVE WHEN THE DEVICE IS ACTIVE !!! *)

(*New dioc data received and the device is active *)
IF in_Dioc_Status.bRxBufferEmpty	OR NOT in_Dioc_Gen_Status.bDeviceActive THEN
	RETURN;
END_IF

(*Process new data *)
CASE Dioc_Register_IN.nRegister			OF



	TP10_R19_CONFIGURATION_SETUP:
		out.nR19_CONFIGURATION_SETUP 		:= Dioc_Register_IN.nValue;

		out.nR19_ROOMTEMPERATURE_AVAILABLE	:= out.nR19_CONFIGURATION_SETUP.0;
		out.nR19_HUMIDITY_AVAILABLE  		:= out.nR19_CONFIGURATION_SETUP.1;
		out.nR19_CO2_AVAILABLE  			:= out.nR19_CONFIGURATION_SETUP.2;
		out.nR19_VOC_AVAILABLE  			:= out.nR19_CONFIGURATION_SETUP.3;
		out.nR19_CO_AVAILABLE  				:= out.nR19_CONFIGURATION_SETUP.4;
		out.nR19_PRESSURE_AVAILABLE  		:= out.nR19_CONFIGURATION_SETUP.5;
		out.nR19_REFPRESSURE_AVAILABLE  	:= out.nR19_CONFIGURATION_SETUP.6;
		out.nR19_ILLUMINATION_AVAILABLE  	:= out.nR19_CONFIGURATION_SETUP.7;
		out.nR19_TOUCH_AVAILABLE  			:= out.nR19_CONFIGURATION_SETUP.8;
		out.nR19_PROXIMITY_AVAILABLE  		:= out.nR19_CONFIGURATION_SETUP.9;
		out.nR19_HAPTIC_AVAILABLE  			:= out.nR19_CONFIGURATION_SETUP.10;
		out.nR19_RGB_AVAILABLE  			:= out.nR19_CONFIGURATION_SETUP.11;

	TP10_R20_ROOMTEMPERATURE_SETUP:
		out.nR20_ROOMTEMPERATURE_SETUP := DWORD_TO_REAL(Dioc_Register_IN.nValue);

	TP10_R21_ROOMTEMPERATURE: 				(* 20 *)
		out.nR21_RoomTemperature 			:= F_SCALE_FROM_DIOC(Dioc_Register_IN.nValue, 0, 4095, -20, 120, -20);

	TP10_R22_ROOM_HUMIDITY_SETUP:
		out.nR22_ROOM_HUMIDITY_SETUP := DWORD_TO_REAL(Dioc_Register_IN.nValue);


	TP10_R23_ROOM_HUMIDITY:
		out.nR23_ROOM_HUMIDITY 			:= F_SCALE_FROM_DIOC(Dioc_Register_IN.nValue, 0, 4095, 0, 100, 0);

	TP10_R24_CO2_SETUP:
		out.nR24_CO2_SETUP 	:= DWORD_TO_REAL(Dioc_Register_IN.nValue);

	TP10_R25_CO2:
		IF ( in_Dioc_Gen_Status.dtR04_VersionHW >= d#2018-06-11 ) AND ( in_Dioc_Gen_Status.dtR05_VersionSW >= d#2018-07-23 ) THEN
			(*new eCO2 sensors*)
			out.nR25_CO2		:= DWORD_TO_REAL(Dioc_Register_IN.nValue);
		ELSE
			(*old eCO2 sensors, correcton on measurement*)
			out.nR25_CO2 		:= DWORD_TO_REAL(267 + Dioc_Register_IN.nValue /3);
		END_IF

	TP10_R26_VOC_SETUP:
		out.nR26_VOC_SETUP := DWORD_TO_REAL(Dioc_Register_IN.nValue);

	TP10_R27_VOC:
		out.nR27_VOC 		:= DWORD_TO_REAL(Dioc_Register_IN.nValue);

	TP10_R28_VOC_BASELINE_L_SETUP:
			out.nR28_VOC_BASELINE_L_SETUP := Dioc_Register_IN.nValue;
			out.br29_VOC_BASELINE_VALID := TRUE;

	TP10_R29_VOC_BASELINE_H_SETUP:
			out.nR29_VOC_BASELINE_H_SETUP := Dioc_Register_IN.nValue;
			in.bR28_VOC_Baseline_L_REQ := TRUE;

	TP10_R34_ROOM_ILLUMINATION_SETUP:
		out.nR34_ROOM_ILLUMINATION_SETUP 		:= DWORD_TO_REAL(Dioc_Register_IN.nValue);

	TP10_R35_ROOM_ILLUMINATION_LUXL_VALUE:
		out.nR35_ROOM_ILLUMINATION_LUXL_VALUE 	:= SEL(Dioc_Register_IN.nValue.11,0,2) + SEL(Dioc_Register_IN.nValue.10,0,1) +SEL(Dioc_Register_IN.nValue.9,0,0.5) +SEL(Dioc_Register_IN.nValue.8,0,0.25);

	TP10_R36_ROOM_ILLUMINATION_LUXH_VALUE:
		out.nR36_ROOM_ILLUMINATION_LUXH_VALUE 	:= DWORD_TO_REAL(Dioc_Register_IN.nValue);
		in.bR35_LUX_L := TRUE;

	TP10_R37_ROOM_ILLUMINATION_IRL_VALUE:
		out.nR37_ROOM_ILLUMINATION_IRL_VALUE 	:=  SEL(Dioc_Register_IN.nValue.11,0,2) + SEL(Dioc_Register_IN.nValue.10,0,1) +SEL(Dioc_Register_IN.nValue.9,0,0.5) +SEL(Dioc_Register_IN.nValue.8,0,0.25);

	TP10_R38_ROOM_ILLUMINATION_IRH_VALUE:
		out.nR38_ROOM_ILLUMINATION_IRH_VALUE 	:= DWORD_TO_REAL(Dioc_Register_IN.nValue);
		in.bR37_IR_L := TRUE;

	TP10_R50_TOUCH_BUTTON_STATUS: (* if the received value is possible, use it, else, request it again. *)
		out.nR50_TouchButtonStatus			:= Dioc_Register_IN.nValue;
		IF 	(out.nR50_TouchButtonStatus.10 OR out.nR50_TouchButtonStatus.11) AND (iNoButtonParity > 0) THEN (* nieuwe versie met pariteit*)
			iNoButtonParity := iNoButtonParity - 1;
		END_IF;

		IF 	(NOT out.nR50_TouchButtonStatus.10) AND (NOT  out.nR50_TouchButtonStatus.11) AND (iNoButtonParity < 100) THEN (* nieuwe versie met pariteit*)
			iNoButtonParity := iNoButtonParity + 1;
		END_IF;

		IF iNoButtonParity < 10 THEN
			IF 	out.nR50_TouchButtonStatus = 2048 OR out.nR50_TouchButtonStatus = 1025 OR out.nR50_TouchButtonStatus = 1026 OR out.nR50_TouchButtonStatus = 1028 OR out.nR50_TouchButtonStatus = 1032 OR out.nR50_TouchButtonStatus = 1040 OR
		 		out.nR50_TouchButtonStatus = 1056 OR  out.nR50_TouchButtonStatus = 1088 OR out.nR50_TouchButtonStatus = 1152 OR out.nR50_TouchButtonStatus = 1280 OR out.nR50_TouchButtonStatus = 1536 THEN

				out.bR50_TouchButton01				:= out.nR50_TouchButtonStatus.0;
				out.bR50_TouchButton02				:= out.nR50_TouchButtonStatus.1;
				out.bR50_TouchButton03				:= out.nR50_TouchButtonStatus.2;
				out.bR50_TouchButton04				:= out.nR50_TouchButtonStatus.3;
				out.bR50_TouchButton05				:= out.nR50_TouchButtonStatus.4;
				out.bR50_TouchButton06				:= out.nR50_TouchButtonStatus.5;
				out.bR50_TouchButton07				:= out.nR50_TouchButtonStatus.6;
				out.bR50_TouchButton08				:= out.nR50_TouchButtonStatus.7;
				out.bR50_TouchButton09				:= out.nR50_TouchButtonStatus.8;
				out.bR50_TouchButton10				:= out.nR50_TouchButtonStatus.9;
			ELSE
				(*re-request the value*)
				in.bR50_TouchButtonStatus := TRUE;
			END_IF;

		ELSE (* versie zonder Pariteitsbits*)
			IF 	out.nR50_TouchButtonStatus = 0 OR out.nR50_TouchButtonStatus = 1 OR out.nR50_TouchButtonStatus = 2 OR out.nR50_TouchButtonStatus = 4 OR out.nR50_TouchButtonStatus = 8 OR out.nR50_TouchButtonStatus = 16 OR
		 		out.nR50_TouchButtonStatus = 32 OR  out.nR50_TouchButtonStatus = 64 OR out.nR50_TouchButtonStatus = 128 OR out.nR50_TouchButtonStatus = 256 OR out.nR50_TouchButtonStatus = 512 THEN

				out.bR50_TouchButton01				:= out.nR50_TouchButtonStatus.0;
				out.bR50_TouchButton02				:= out.nR50_TouchButtonStatus.1;
				out.bR50_TouchButton03				:= out.nR50_TouchButtonStatus.2;
				out.bR50_TouchButton04				:= out.nR50_TouchButtonStatus.3;
				out.bR50_TouchButton05				:= out.nR50_TouchButtonStatus.4;
				out.bR50_TouchButton06				:= out.nR50_TouchButtonStatus.5;
				out.bR50_TouchButton07				:= out.nR50_TouchButtonStatus.6;
				out.bR50_TouchButton08				:= out.nR50_TouchButtonStatus.7;
				out.bR50_TouchButton09				:= out.nR50_TouchButtonStatus.8;
				out.bR50_TouchButton10				:= out.nR50_TouchButtonStatus.9;
			ELSE
				(*re-request the value*)
				in.bR50_TouchButtonStatus := TRUE;
			END_IF;
		END_IF;


	TP10_R51_TOUCH_LED_STATUS:				(* 51 *)
		byParity := INT_TO_BYTE(BOOL_TO_INT(Dioc_Register_IN.nValue.0) + BOOL_TO_INT(Dioc_Register_IN.nValue.1) + BOOL_TO_INT(Dioc_Register_IN.nValue.2) + BOOL_TO_INT(Dioc_Register_IN.nValue.3) + BOOL_TO_INT(Dioc_Register_IN.nValue.4) + BOOL_TO_INT(Dioc_Register_IN.nValue.5) + BOOL_TO_INT(Dioc_Register_IN.nValue.6) + BOOL_TO_INT(Dioc_Register_IN.nValue.7) + BOOL_TO_INT(Dioc_Register_IN.nValue.8) + BOOL_TO_INT(Dioc_Register_IN.nValue.9));
		IF Dioc_Register_IN.nValue.10 = byParity.0 AND Dioc_Register_IN.nValue.11 <> byParity.0 OR (iNoButtonParity >= 10) THEN
			out.nR51_TouchLedStatus				:= Dioc_Register_IN.nValue;
		END_IF;

	TP10_R52_TOUCH_LED_MASK:				(* 52 *)
		byParity := INT_TO_BYTE(BOOL_TO_INT(Dioc_Register_IN.nValue.0) + BOOL_TO_INT(Dioc_Register_IN.nValue.1) + BOOL_TO_INT(Dioc_Register_IN.nValue.2) + BOOL_TO_INT(Dioc_Register_IN.nValue.3) + BOOL_TO_INT(Dioc_Register_IN.nValue.4) + BOOL_TO_INT(Dioc_Register_IN.nValue.5) + BOOL_TO_INT(Dioc_Register_IN.nValue.6) + BOOL_TO_INT(Dioc_Register_IN.nValue.7) + BOOL_TO_INT(Dioc_Register_IN.nValue.8) + BOOL_TO_INT(Dioc_Register_IN.nValue.9));
		IF Dioc_Register_IN.nValue.10 = byParity.0 AND Dioc_Register_IN.nValue.11 <> byParity.0 OR (iNoButtonParity >= 10) THEN
			out.nR52_TouchLedMask				:= Dioc_Register_IN.nValue;
		END_IF;

	TP10_R57_HAPTIC_INTENSITY:
		;


	ELSE;
END_CASE
END_ACTION

ACTION Restart:
(* Invalidate previous status with something impossible and not dangerous, must be something that will be updated by the cycle *)
stDeviceDataInPrevious.nR51_TouchLedStatus := 16500;
stDeviceDataInPrevious.NR83_ButtonSensitivity := 0;

out := outRef;
(* invalidate out feedback used in the send conditions *)
iRefreshCycles := 0;

(* Re-set the status of the leds *)
(*
in.nR51_TouchLedStatus		:= out.nR51_TouchLedStatus;
in.nR52_TouchLedMask		:= out.nR52_TouchLedMask;
*)

(* Acknowledge *)
bRestarted := FALSE;
END_ACTION

ACTION Send:
(* !!! ONLY ACTIVE WHEN THE DEVICE IS ACTIVE !!! *)

(*
	is the device active *)
IF NOT in_Dioc_Gen_Status.bDeviceActive THEN
	(*reset all saved values*)
	RETURN;
END_IF



(*
	New dioc data received ? *)
IF MEMCMP(ADR(stDeviceDataInPrevious), ADR(in), SIZEOF(stDeviceDataInPrevious)) = 0 THEN RETURN; END_IF;

nTemp := MEMCMP(ADR(stDeviceDataInPrevious), ADR(in), SIZEOF(stDeviceDataInPrevious));

(*opbouw RGB*)
in.nR61_RGB_MSB.0 := in.nR61_RGB_RED.4;
in.nR61_RGB_MSB.1 := in.nR61_RGB_RED.5;
in.nR61_RGB_MSB.2 := in.nR61_RGB_RED.6;
in.nR61_RGB_MSB.3 := in.nR61_RGB_RED.7;
in.nR61_RGB_MSB.4 := in.nR61_RGB_GREEN.4;
in.nR61_RGB_MSB.5 := in.nR61_RGB_GREEN.5;
in.nR61_RGB_MSB.6 := in.nR61_RGB_GREEN.6;
in.nR61_RGB_MSB.7 := in.nR61_RGB_GREEN.7;
in.nR61_RGB_MSB.8 := in.nR61_RGB_BLUE.4;
in.nR61_RGB_MSB.9 := in.nR61_RGB_BLUE.5;
in.nR61_RGB_MSB.10 := in.nR61_RGB_BLUE.6;
in.nR61_RGB_MSB.11 := in.nR61_RGB_BLUE.7;

in.nR62_RGB_LSB.0 := in.nR61_RGB_RED.0;
in.nR62_RGB_LSB.1 := in.nR61_RGB_RED.1;
in.nR62_RGB_LSB.2 := in.nR61_RGB_RED.2;
in.nR62_RGB_LSB.3 := in.nR61_RGB_RED.3;
in.nR62_RGB_LSB.4 := in.nR61_RGB_GREEN.0;
in.nR62_RGB_LSB.5 := in.nR61_RGB_GREEN.1;
in.nR62_RGB_LSB.6 := in.nR61_RGB_GREEN.2;
in.nR62_RGB_LSB.7 := in.nR61_RGB_GREEN.3;
in.nR62_RGB_LSB.8 := in.nR61_RGB_BLUE.0;
in.nR62_RGB_LSB.9 := in.nR61_RGB_BLUE.1;
in.nR62_RGB_LSB.10 := in.nR61_RGB_BLUE.2;
in.nR62_RGB_LSB.11 := in.nR61_RGB_BLUE.3;

(*
	Handle register handling in the order of priority *)
(* PRIORITY 00: internal commands (eg at startup) *)
(* Test message, highest priority, always send a sync message first *)
nPriority := 0;

(* PRIORITY 01 *)
nPriority := 1;

(* PRIORITY 02 *)
nPriority := 2;
(* PRIORITY 03 *)
nPriority := 3;
IF in.nR51_TouchLedStatus <> stDeviceDataInPrevious.nR51_TouchLedStatus  OR iRefreshCycles = 320 THEN				(* Set touch led status *)
	byParity := INT_TO_BYTE(BOOL_TO_INT(in.nR51_TouchLedStatus.0) + BOOL_TO_INT(in.nR51_TouchLedStatus.1) + BOOL_TO_INT(in.nR51_TouchLedStatus.2) + BOOL_TO_INT(in.nR51_TouchLedStatus.3) + BOOL_TO_INT(in.nR51_TouchLedStatus.4) + BOOL_TO_INT(in.nR51_TouchLedStatus.5) + BOOL_TO_INT(in.nR51_TouchLedStatus.6) + BOOL_TO_INT(in.nR51_TouchLedStatus.7) + BOOL_TO_INT(in.nR51_TouchLedStatus.8) + BOOL_TO_INT(in.nR51_TouchLedStatus.9));
	bTxBuffer_Write					:= TRUE;
	fbTxBuffer[nPriority](
		IN							:= F_DIOC_20_MESSAGE_OUT(nRegister := TP10_R51_TOUCH_LED_STATUS, nValue := SEL(byParity.0,in.nR51_TouchLedStatus+2048,in.nR51_TouchLedStatus+1024)),
		RD							:= bTxBuffer_Read,			(* Not functional *)
		WD							:= bTxBuffer_Write,
		fifo						:= ADR(TxBuffer[nPriority, 0]));
	IF NOT bTxBuffer_Write			THEN	(* Successfully transferred to the Tx Buffer *)
		stDeviceDataInPrevious.nR51_TouchLedStatus			:= in.nR51_TouchLedStatus;
	END_IF
END_IF

IF in.nR52_TouchLedMask <> stDeviceDataInPrevious.nR52_TouchLedMask  OR iRefreshCycles = 360 THEN	(* Set touch led mask *)
	byParity := INT_TO_BYTE(BOOL_TO_INT(in.nR52_TouchLedMask.0) + BOOL_TO_INT(in.nR52_TouchLedMask.1) + BOOL_TO_INT(in.nR52_TouchLedMask.2) + BOOL_TO_INT(in.nR52_TouchLedMask.3) + BOOL_TO_INT(in.nR52_TouchLedMask.4) + BOOL_TO_INT(in.nR52_TouchLedMask.5) + BOOL_TO_INT(in.nR52_TouchLedMask.6) + BOOL_TO_INT(in.nR52_TouchLedMask.7) + BOOL_TO_INT(in.nR52_TouchLedMask.8) + BOOL_TO_INT(in.nR52_TouchLedMask.9));
	bTxBuffer_Write					:= TRUE;
	fbTxBuffer[nPriority](
		IN							:= F_DIOC_20_MESSAGE_OUT(nRegister := TP10_R52_TOUCH_LED_MASK, nValue := SEL(byParity.0,in.nR52_TouchLedMask+2048,in.nR52_TouchLedMask+1024)),
		RD							:= bTxBuffer_Read,			(* Not functional *)
		WD							:= bTxBuffer_Write,
		fifo						:= ADR(TxBuffer[nPriority, 0]));
	IF NOT bTxBuffer_Write			THEN	(* Successfully transferred to the Tx Buffer *)
		stDeviceDataInPrevious.nR52_TouchLedMask			:= in.nR52_TouchLedMask;
	END_IF
END_IF
(* PRIORITY 04 *)
nPriority := 4;
IF in.NR83_ButtonSensitivity <> stDeviceDataInPrevious.NR83_ButtonSensitivity THEN	(* write the button sensitivity*)
	IF ((in.NR83_ButtonSensitivity >0) AND (in.NR83_ButtonSensitivity <100)) THEN
		bTxBuffer_Write					:= TRUE;
		fbTxBuffer[nPriority](
			IN							:= F_DIOC_20_MESSAGE_OUT(nRegister := TP10_R83_BUTTON_SENSITIVITY, nValue := in.NR83_ButtonSensitivity),
			RD							:= bTxBuffer_Read,			(* Not functional *)
			WD							:= bTxBuffer_Write,
			fifo						:= ADR(TxBuffer[nPriority, 0]));
		IF NOT bTxBuffer_Write			THEN	(* Successfully transferred to the Tx Buffer *)
			stDeviceDataInPrevious.NR83_ButtonSensitivity := in.NR83_ButtonSensitivity;
		END_IF
	END_IF
END_IF

(* PRIORITY 05 *)
nPriority := 5;

(* PRIORITY 06 *)
nPriority := 6;

(* PRIORITY 07 *)
nPriority := 7;

IF in.bR19_Configuration_Setup THEN		(* Request configuration setup*)
	fbTxBuffer[nPriority](
		IN							:= F_DIOC_20_MESSAGE_OUT(nRegister := DIOC_R01_REGISTER_REQUEST, nValue := TP10_R19_CONFIGURATION_SETUP),
		RD							:= bTxBuffer_Read,			(* Not functional *)
		WD							:= in.bR19_Configuration_Setup,
		fifo						:= ADR(TxBuffer[nPriority, 0]));
END_IF

IF in.bR20_Room_Temperature_Setup			THEN		(* Request room temperature setup*)
	bTxBuffer_Write					:= TRUE;
	fbTxBuffer[nPriority](
		IN							:= F_DIOC_20_MESSAGE_OUT(nRegister :=DIOC_R01_REGISTER_REQUEST  , nValue := TP10_R20_ROOMTEMPERATURE_SETUP),
		RD							:= bTxBuffer_Read,			(* Not functional *)
		WD							:= bTxBuffer_Write,
		fifo						:= ADR(TxBuffer[nPriority, 0]));
	in.bR20_Room_Temperature_Setup := FALSE;
END_IF

IF in.bR21_Room_Temperature			THEN		(* Request room temperature *)
	(*out.nR20_Room_Temperature		:= -1;*) (*TV // not necesairy, down point in trending software*)
	fbTxBuffer[nPriority](
		IN							:= F_DIOC_20_MESSAGE_OUT(nRegister := DIOC_R01_REGISTER_REQUEST, nValue := TP10_R21_ROOMTEMPERATURE),
		RD							:= bTxBuffer_Read,			(* Not functional *)
		WD							:= in.bR21_Room_Temperature,
		fifo						:= ADR(TxBuffer[nPriority, 0]));
END_IF

IF in.bR22_Room_Humidity_Setup			THEN		(* Request room temperature setup*)
	fbTxBuffer[nPriority](
		IN							:= F_DIOC_20_MESSAGE_OUT(nRegister :=DIOC_R01_REGISTER_REQUEST  , nValue := TP10_R22_ROOM_HUMIDITY_SETUP),
		RD							:= bTxBuffer_Read,			(* Not functional *)
		WD							:= in.bR22_Room_Humidity_Setup,
		fifo						:= ADR(TxBuffer[nPriority, 0]));
END_IF

IF in.bR24_CO2_Setup			THEN		(* Request CO2 setup*)
	fbTxBuffer[nPriority](
		IN							:= F_DIOC_20_MESSAGE_OUT(nRegister :=DIOC_R01_REGISTER_REQUEST  , nValue := TP10_R24_CO2_SETUP),
		RD							:= bTxBuffer_Read,			(* Not functional *)
		WD							:= in.bR24_CO2_Setup,
		fifo						:= ADR(TxBuffer[nPriority, 0]));
END_IF

IF in.bR26_VOC_Setup			THEN		(* Request VOC setup*)
	fbTxBuffer[nPriority](
		IN							:= F_DIOC_20_MESSAGE_OUT(nRegister :=DIOC_R01_REGISTER_REQUEST  , nValue := TP10_R26_VOC_SETUP),
		RD							:= bTxBuffer_Read,			(* Not functional *)
		WD							:= in.bR26_VOC_Setup,
		fifo						:= ADR(TxBuffer[nPriority, 0]));
END_IF

IF in.bR28_VOC_Baseline_L_REQ THEN
	fbTxBuffer[nPriority](
		IN							:= F_DIOC_20_MESSAGE_OUT(nRegister :=DIOC_R01_REGISTER_REQUEST  , nValue := TP10_R28_VOC_BASELINE_L_SETUP),
		RD							:= bTxBuffer_Read,			(* Not functional *)
		WD							:= in.bR28_VOC_Baseline_L_REQ,
		fifo						:= ADR(TxBuffer[nPriority, 0]));
END_IF;

IF in.bR28_VOC_Baseline_L_SEND THEN
	fbTxBuffer[nPriority](
		IN							:= F_DIOC_20_MESSAGE_OUT(nRegister :=TP10_R28_VOC_BASELINE_L_SETUP  , nValue := out.nR28_VOC_BASELINE_L_SETUP),
		RD							:= bTxBuffer_Read,			(* Not functional *)
		WD							:= in.bR28_VOC_Baseline_L_SEND,
		fifo						:= ADR(TxBuffer[nPriority, 0]));
END_IF;

IF in.bR29_VOC_Baseline_H_REQ THEN
	fbTxBuffer[nPriority](
		IN							:= F_DIOC_20_MESSAGE_OUT(nRegister :=DIOC_R01_REGISTER_REQUEST  , nValue := TP10_R29_VOC_BASELINE_H_SETUP),
		RD							:= bTxBuffer_Read,			(* Not functional *)
		WD							:= in.bR29_VOC_BaseLine_H_REQ,
		fifo						:= ADR(TxBuffer[nPriority, 0]));
END_IF;

IF in.bR29_VOC_Baseline_H_SEND THEN
	fbTxBuffer[nPriority](
		IN							:= F_DIOC_20_MESSAGE_OUT(nRegister :=TP10_R29_VOC_BASELINE_H_SETUP  , nValue := out.nR29_VOC_BASELINE_H_SETUP),
		RD							:= bTxBuffer_Read,			(* Not functional *)
		WD							:= in.bR29_VOC_Baseline_H_SEND,
		fifo						:= ADR(TxBuffer[nPriority, 0]));
	in.bR28_VOC_BaseLine_L_SEND := TRUE;
END_IF;

IF in.bR34_LUX_Setup THEN
	fbTxBuffer[nPriority](
		IN							:= F_DIOC_20_MESSAGE_OUT(nRegister :=DIOC_R01_REGISTER_REQUEST  , nValue := TP10_R34_ROOM_ILLUMINATION_SETUP),
		RD							:= bTxBuffer_Read,			(* Not functional *)
		WD							:= in.bR34_LUX_Setup,
		fifo						:= ADR(TxBuffer[nPriority, 0]));
END_IF

IF in.bR35_LUX_L THEN
	fbTxBuffer[nPriority](
		IN							:= F_DIOC_20_MESSAGE_OUT(nRegister :=DIOC_R01_REGISTER_REQUEST  , nValue := TP10_R35_ROOM_ILLUMINATION_LUXL_VALUE),
		RD							:= bTxBuffer_Read,			(* Not functional *)
		WD							:= in.bR35_LUX_L,
		fifo						:= ADR(TxBuffer[nPriority, 0]));
END_IF

IF in.bR36_LUX_H THEN
	fbTxBuffer[nPriority](
		IN							:= F_DIOC_20_MESSAGE_OUT(nRegister :=DIOC_R01_REGISTER_REQUEST  , nValue := TP10_R36_ROOM_ILLUMINATION_LUXH_VALUE),
		RD							:= bTxBuffer_Read,			(* Not functional *)
		WD							:= in.bR36_LUX_H,
		fifo						:= ADR(TxBuffer[nPriority, 0]));
END_IF

IF in.bR37_IR_L THEN
	fbTxBuffer[nPriority](
		IN							:= F_DIOC_20_MESSAGE_OUT(nRegister :=DIOC_R01_REGISTER_REQUEST  , nValue := TP10_R37_ROOM_ILLUMINATION_IRL_VALUE),
		RD							:= bTxBuffer_Read,			(* Not functional *)
		WD							:= in.bR37_IR_L,
		fifo						:= ADR(TxBuffer[nPriority, 0]));
END_IF

IF in.bR38_IR_H THEN
	fbTxBuffer[nPriority](
		IN							:= F_DIOC_20_MESSAGE_OUT(nRegister :=DIOC_R01_REGISTER_REQUEST  , nValue := TP10_R38_ROOM_ILLUMINATION_IRH_VALUE),
		RD							:= bTxBuffer_Read,			(* Not functional *)
		WD							:= in.bR38_IR_H,
		fifo						:= ADR(TxBuffer[nPriority, 0]));
END_IF

IF in.bR50_TouchButtonStatus OR iRefreshCycles = 120		THEN		(* Request touch button status *)
	fbTxBuffer[nPriority](
		IN							:= F_DIOC_20_MESSAGE_OUT(nRegister := DIOC_R01_REGISTER_REQUEST, nValue := TP10_R50_TOUCH_BUTTON_STATUS),
		RD							:= bTxBuffer_Read,			(* Not functional *)
		WD							:= in.bR50_TouchButtonStatus,
		fifo						:= ADR(TxBuffer[nPriority, 0]));
END_IF

IF in.bR51_TouchLedStatus OR iRefreshCycles = 40		THEN		(* Request touch led status *)
	out.nR51_TouchLedStatus			:= 0;
	fbTxBuffer[nPriority](
		IN							:= F_DIOC_20_MESSAGE_OUT(nRegister := DIOC_R01_REGISTER_REQUEST, nValue := TP10_R51_TOUCH_LED_STATUS),
		RD							:= bTxBuffer_Read,			(* Not functional *)
		WD							:= in.bR51_TouchLedStatus,
		fifo						:= ADR(TxBuffer[nPriority, 0]));
END_IF

IF in.bR52_TouchLedMaskStatus OR iRefreshCycles = 40		THEN		(* Request touch led status *)
	out.nR52_TouchLedMask			:= 0;
	fbTxBuffer[nPriority](
		IN							:= F_DIOC_20_MESSAGE_OUT(nRegister := DIOC_R01_REGISTER_REQUEST, nValue := TP10_R52_TOUCH_LED_MASK),
		RD							:= bTxBuffer_Read,			(* Not functional *)
		WD							:= in.bR52_TouchLedMaskStatus,
		fifo						:= ADR(TxBuffer[nPriority, 0]));
END_IF

IF in.nR53_LED_Intensity_Max <> stDeviceDataInPrevious.nR53_LED_Intensity_Max 	OR iRefreshCycles = 320 THEN	(*TV160314A // Write led intensity *)
	bTxBuffer_Write					:= TRUE;
	fbTxBuffer[nPriority](
		IN							:= F_DIOC_20_MESSAGE_OUT(nRegister :=TP10_R53_LED_Intensity_Max  , nValue := in.nR53_LED_Intensity_Max),
		RD							:= bTxBuffer_Read,			(* Not functional *)
		WD							:= bTxBuffer_Write,
		fifo						:= ADR(TxBuffer[nPriority, 0]));
	stDeviceDataInPrevious.nR53_LED_Intensity_Max := in.nR53_LED_Intensity_Max;
END_IF

IF in.bR57_HapticIntensity OR (in.nR57_HapticIntensity <> stDeviceDataInPrevious.nR57_HapticIntensity)	 OR iRefreshCycles = 240 THEN	(*TV160314A // haptic intensity *)
	bTxBuffer_Write					:= TRUE;
	fbTxBuffer[nPriority](
		IN							:= F_DIOC_20_MESSAGE_OUT(nRegister := TP10_R57_HAPTIC_INTENSITY, nValue := in.nR57_HapticIntensity),
		RD							:= bTxBuffer_Read,			(* Not functional *)
		WD							:= bTxBuffer_Write,
		fifo						:= ADR(TxBuffer[nPriority, 0]));
	stDeviceDataInPrevious.nR57_HapticIntensity := in.nR57_HapticIntensity;
	in.bR57_HapticIntensity := FALSE;
END_IF

IF NOT (in.nR60_RGB_LED_SETUP = stDeviceDataInPrevious.nR60_RGB_LED_SETUP ) THEN
	bTxBuffer_Write					:= TRUE;
	fbTxBuffer[nPriority](
		IN							:= F_DIOC_20_MESSAGE_OUT(nRegister :=TP10_R60_RGB_LED_SETUP  , nValue := in.nR60_RGB_LED_SETUP),
		RD							:= bTxBuffer_Read,			(* Not functional *)
		WD							:= bTxBuffer_Write,
		fifo						:= ADR(TxBuffer[nPriority, 0]));
	stDeviceDataInPrevious.nR60_RGB_LED_SETUP := in.nR60_RGB_LED_SETUP;
END_IF

IF NOT (stDeviceDataInPrevious.nR61_RGB_MSB = in.nR61_RGB_MSB) OR iRefreshCycles = 160	THEN	(*HS16/10/26 // Write RGB led intensity most significant bits *)
	bTxBuffer_Write					:= TRUE;
	fbTxBuffer[nPriority](
		IN							:= F_DIOC_20_MESSAGE_OUT(nRegister :=TP10_R61_RGB_MSB  , nValue := in.nR61_RGB_MSB),
		RD							:= bTxBuffer_Read,			(* Not functional *)
		WD							:= bTxBuffer_Write,
		fifo						:= ADR(TxBuffer[nPriority, 0]));
	stDeviceDataInPrevious.nR61_RGB_MSB := in.nR61_RGB_MSB;
END_IF

IF NOT (stDeviceDataInPrevious.nR62_RGB_LSB = in.nR62_RGB_LSB) OR iRefreshCycles = 200 THEN	(*HS16/10/26 // Write RGB led intensity least significant bits *)
	bTxBuffer_Write					:= TRUE;
	fbTxBuffer[nPriority](
		IN							:= F_DIOC_20_MESSAGE_OUT(nRegister :=TP10_R62_RGB_LSB  , nValue := in.nR62_RGB_LSB),
		RD							:= bTxBuffer_Read,			(* Not functional *)
		WD							:= bTxBuffer_Write,
		fifo						:= ADR(TxBuffer[nPriority, 0]));
	stDeviceDataInPrevious.nR62_RGB_LSB := in.nR62_RGB_LSB;
END_IF

IF ((in.NR82_Temp_offset<>stDeviceDataInPrevious.NR82_Temp_offset) OR (in.bR82_Temp_offset)) THEN
	bTxBuffer_Write					:= TRUE;
	fbTxBuffer[nPriority](
		IN							:= F_DIOC_20_MESSAGE_OUT(nRegister :=TP10_R82_TEMP_OFFSET  , nValue := in.NR82_Temp_offset),
		RD							:= bTxBuffer_Read,			(* Not functional *)
		WD							:= bTxBuffer_Write,
		fifo						:= ADR(TxBuffer[nPriority, 0]));
	stDeviceDataInPrevious.NR82_Temp_offset := in.NR82_Temp_offset;
	in.bR82_Temp_offset := FALSE;
END_IF

IF ((in.NR86_Temp_offset<>stDeviceDataInPrevious.NR86_Temp_offset) OR (in.bR86_Temp_offset)) THEN
	bTxBuffer_Write					:= TRUE;
	fbTxBuffer[nPriority](
		IN							:= F_DIOC_20_MESSAGE_OUT(nRegister :=TP10_R86_TEMP_OFFSET  , nValue := in.NR86_Temp_offset),
		RD							:= bTxBuffer_Read,			(* Not functional *)
		WD							:= bTxBuffer_Write,
		fifo						:= ADR(TxBuffer[nPriority, 0]));
	stDeviceDataInPrevious.NR86_Temp_offset := in.NR86_Temp_offset;
	in.bR86_Temp_offset := FALSE;
END_IF

(* PRIORITY 08 *)
nPriority := 8;

IF NOT (stDeviceDataInPrevious.nR20_ROOMTEMPERATURE_SETUP = in.nR20_ROOMTEMPERATURE_SETUP) THEN
	bTxBuffer_Write					:= TRUE;
	fbTxBuffer[nPriority](
		IN							:= F_DIOC_20_MESSAGE_OUT(nRegister :=TP10_R20_ROOMTEMPERATURE_SETUP  , nValue := in.nR20_ROOMTEMPERATURE_SETUP),
		RD							:= bTxBuffer_Read,			(* Not functional *)
		WD							:= bTxBuffer_Write,
		fifo						:= ADR(TxBuffer[nPriority, 0]));
	stDeviceDataInPrevious.nR20_ROOMTEMPERATURE_SETUP := in.nR20_ROOMTEMPERATURE_SETUP;
END_IF

IF NOT (stDeviceDataInPrevious.nR22_ROOM_HUMIDITY_SETUP = in.nR22_ROOM_HUMIDITY_SETUP) THEN
	bTxBuffer_Write					:= TRUE;
	fbTxBuffer[nPriority](
		IN							:= F_DIOC_20_MESSAGE_OUT(nRegister :=TP10_R22_ROOM_HUMIDITY_SETUP  , nValue := in.nR22_ROOM_HUMIDITY_SETUP),
		RD							:= bTxBuffer_Read,			(* Not functional *)
		WD							:= bTxBuffer_Write,
		fifo						:= ADR(TxBuffer[nPriority, 0]));
	stDeviceDataInPrevious.nR22_ROOM_HUMIDITY_SETUP := in.nR22_ROOM_HUMIDITY_SETUP;
END_IF

IF NOT (stDeviceDataInPrevious.nR24_CO2_SETUP = in.nR24_CO2_SETUP) THEN
	bTxBuffer_Write					:= TRUE;
	fbTxBuffer[nPriority](
		IN							:= F_DIOC_20_MESSAGE_OUT(nRegister :=TP10_R24_CO2_SETUP  , nValue := in.nR24_CO2_SETUP),
		RD							:= bTxBuffer_Read,			(* Not functional *)
		WD							:= bTxBuffer_Write,
		fifo						:= ADR(TxBuffer[nPriority, 0]));
	stDeviceDataInPrevious.nR24_CO2_SETUP := in.nR24_CO2_SETUP;
END_IF

IF NOT (stDeviceDataInPrevious.nR26_VOC_SETUP = in.nR26_VOC_SETUP) THEN
	bTxBuffer_Write					:= TRUE;
	fbTxBuffer[nPriority](
		IN							:= F_DIOC_20_MESSAGE_OUT(nRegister :=TP10_R26_VOC_SETUP  , nValue := in.nR26_VOC_SETUP),
		RD							:= bTxBuffer_Read,			(* Not functional *)
		WD							:= bTxBuffer_Write,
		fifo						:= ADR(TxBuffer[nPriority, 0]));
	stDeviceDataInPrevious.nR26_VOC_SETUP := in.nR26_VOC_SETUP;
END_IF

IF NOT (stDeviceDataInPrevious.nR34_ROOM_ILLUMINATION_SETUP = in.nR34_ROOM_ILLUMINATION_SETUP) THEN
	bTxBuffer_Write					:= TRUE;
	fbTxBuffer[nPriority](
		IN							:= F_DIOC_20_MESSAGE_OUT(nRegister :=TP10_R34_ROOM_ILLUMINATION_SETUP  , nValue := in.nR34_ROOM_ILLUMINATION_SETUP),
		RD							:= bTxBuffer_Read,			(* Not functional *)
		WD							:= bTxBuffer_Write,
		fifo						:= ADR(TxBuffer[nPriority, 0]));
	stDeviceDataInPrevious.nR34_ROOM_ILLUMINATION_SETUP := in.nR34_ROOM_ILLUMINATION_SETUP;
END_IF
END_ACTION

ACTION Startup:
iRefreshCycles := 0;
END_ACTION

END_FUNCTION_BLOCK

// POUs/DIOC/TP10/_Internal/FB_TP10_COMM
FUNCTION_BLOCK FB_TP10_COMM
VAR_INPUT
	in									: ST_TP10_IN;
	iPowerCycleGroup					: INT;
END_VAR
VAR_OUTPUT
	out									: ST_TP10_OUT;
	nError								: E_TP10_ERROR;
END_VAR
VAR CONSTANT
	TYPE_ID								: DWORD		:= 1;		(* Device identifier *)
	DEVICE_CHARGE_TIME					: TIME 		:= T#2s;	(* Optional charge time *)
	DIOC_LENGTH							: INT 		:= 21;		(* Dioc protocol length *)
	SYNC_MESSAGE							: DWORD		:= 2#0000_0000_000_1_1010_1010_1010_1111111_0;		(* Sync request = request type id *)
	SYNC_MESSAGE_HIGH					: DWORD		:= 2#0000_0000_000_1_0101_0101_0101_0101010_0;		(* Sync request = request type id *)
	DEVICE_CALIBRATION_TIME				: TIME		:= t#5s;	(* Time for calibrating touch buttons *)
	DEVICE_CALIBRATION_LED_DELAY		: TIME		:= t#250ms;	(* Running leds at calibration time *)
END_VAR
VAR
(* TC3 attribute, will be ignored by TC2 *)
{attribute 'hide_all_locals'}
(* TC2 attribute, will be ignored by TC3 *)
{library private}
	(*
		Startup list *)
	bStartup							: BOOL 		:= TRUE;
	bRestarted							: BOOL;					(* Device hardware restart detected by dioc *)

	(* Buffer communication *)
	Dioc_Register_IN					: ST_DIOC_REGISTER;		(* Message retrieved from buffer *)
	bRxBuffer_Read						: BOOL;
	bRxBuffer_Write						: BOOL;

	(* Fifo Buffers *)
	RxBuffer							: ARRAY[0..DIOC_RXTX_BUFFERSIZE] OF A_DIOC_MESSAGE;	(* 1 message queue *)
	TxBuffer							: ARRAY[0..DIOC_MAXPRIORITY, 0..DIOC_RXTX_BUFFERSIZE] OF A_DIOC_MESSAGE;	(* 1 message queue / priority, HIGHEST: 0 = internal priority *)

	(* Fifo Buffer handlers *)
	fbRxBuffer							: FB_DIOC_FIFO;									(* 1 message queue *)
	fbTxBuffer							: ARRAY[0..DIOC_MAXPRIORITY] OF FB_DIOC_FIFO;	(* 1 message queue / priority *)

	(* Dioc base communication layer *)
	fbDioc								: FB_DIOC;
	(* Device general register handling *)
	fbDioc_Gen							: FB_DIOC_GEN;
	(* Device specific register handling *)
	fbDioc_Tp10							: FB_DIOC_TP10;

	(* State machine *)
	nSm									: E_TP10;

	i									: INT;

	(*Internal tp10 commands*)
	(*This structure give the possibility to sperate the incomming commands from the internal commands during calibration*)
	_in									: ST_TP10_IN;

END_VAR

(*
	startup *)
IF bStartup THEN Startup(); END_IF
fbDioc.iPowerCycleGroup := iPowerCycleGroup;
(*
	Get next message from message queue *)
bRxBuffer_Read				:= NOT fbDioc.Out.bRxBufferEmpty;
fbRxBuffer(
	RD						:= bRxBuffer_Read,
	WD						:= bRxBuffer_Write,				(* Not functional *)
	fifo					:= ADR(RxBuffer));
Dioc_Register_IN := F_DIOC_20_MESSAGE_IN(fbRxBuffer.OUT);

(* Device Dioc base register handling and startup parameter loading *)
fbDioc_Gen(
	in						:= in.DIOC_Gen,
	in_Dioc_Status			:= fbDioc.Out,
	TYPE_ID					:= TYPE_ID,
	Dioc_Register_IN		:= Dioc_Register_IN,
	RxBuffer				:= RxBuffer,
	TxBuffer				:= TxBuffer,
	fbRxBuffer				:= fbRxBuffer,
	fbTxBuffer				:= fbTxBuffer,
	arrstStartupParameter	:= in.DIOC_TP10.arrstStartupParameter,
	bRestarted				:= bRestarted,
	out						=> out.DIOC_Gen,
	nError					=>
	);
in.DIOC_Gen 				:= fbDioc_Gen.in;				(* Copy possibly changed inputs back to upper level *)

(* Device specific register handling *)
(*lock external commands during calibration*)
IF nSm<>TP10_CALIBRATED THEN
	fbDioc_Tp10.in:=in.DIOC_TP10;
ELSE
	fbDioc_Tp10.in:=in.DIOC_TP10;
END_IF

fbDioc_Tp10(
	in						:= , (*Written above*)
	in_Dioc_Status			:= fbDioc.Out,
	in_Dioc_Gen_Status		:= fbDioc_Gen.Out,
	Dioc_Register_IN		:= Dioc_Register_IN,
	RxBuffer				:= RxBuffer,
	TxBuffer				:= TxBuffer,
	fbRxBuffer				:= fbRxBuffer,
	fbTxBuffer				:= fbTxBuffer,
	bRestarted				:= bRestarted,
	out						=> out.DIOC_TP10,
	nError					=>
	);

IF nSm=TP10_CALIBRATED THEN
	in.DIOC_Tp10				:= fbDioc_Tp10.in;				(* Copy possibly changed inputs back to upper level *)
END_IF
(*
	Dioc communication layer *)
fbDioc.in.bEnable			:= in.bEnable;	(* Debug *)
fbDioc(
	DEVICE_CHARGE_TIME		:= DEVICE_CHARGE_TIME,
	DIOC_LENGTH				:= DIOC_LENGTH,
	RxBuffer				:= RxBuffer,
	TxBuffer				:= TxBuffer,
	fbRxBuffer				:= fbRxBuffer,
	fbTxBuffer				:= fbTxBuffer,
	Out						=>
	);

(*
	State machine *)
IF NOT fbDioc_Gen.out.bDeviceActive	THEN
	nSm								:= TP10_INIT;
END_IF

CASE nSm					OF

	TP10_INIT:
		(* Startup if device is active *)
		IF NOT fbDioc_Gen.out.bDeviceActive		THEN
			nSm						:= TP10_START_CALIBRATION;
		END_IF

	TP10_START_CALIBRATION:
		(* disable leds *)
		nSm							:= TP10_SET_LED;

	TP10_SET_LED:
		(* rainbow mode *)
		(*in.DIOC_TP10.nR60_RGB_LED_SETUP := 2;*)
		nSm							:= TP10_WAIT_STARTUP;

	TP10_WAIT_STARTUP:
		IF fbDioc_Gen.out.bDeviceActive	THEN
			nSm						:= TP10_RESET_LED;
		END_IF

	TP10_RESET_LED:
		(*_in.DIOC_TP10.nR51_TouchLedStatus := 2048;*)
		(*in.DIOC_TP10.nR60_RGB_LED_SETUP := 0;*)
		nSm							:= TP10_CALIBRATED;

	TP10_CALIBRATED:
		(*in.DIOC_TP10.nR60_RGB_LED_SETUP := 0*);

	ELSE;

END_CASE
out.DIOC_TP10.bCalibrationFinished	:= nSm=TP10_CALIBRATED;

(*
	First loop finished *)
bStartup 					:= FALSE;

ACTION Startup:
(*
	Startup parameters, can be set here or default in the in struct *) 

(* Reset parameters
FOR i := 1 TO DIOC_NOOFSTARTUPPARAMETERS DO
	in.arrstStartupParameter[i].nRegister		:= 255;	(* Set to invalid *)
	arrstStartupParameter[i].nValue			:= 0;
END_FOR *)

(* Test Set parameters, switch relays
arrstStartupParameter[1].nRegister			:= 25;
arrstStartupParameter[1].nValue				:= 3;
arrstStartupParameter[2].nRegister			:= 32;
arrstStartupParameter[2].nValue				:= 3;
arrstStartupParameter[3].nRegister			:= 52;
arrstStartupParameter[3].nValue				:= 1;
arrstStartupParameter[4].nRegister			:= 25;
arrstStartupParameter[4].nValue				:= 1;
arrstStartupParameter[5].nRegister			:= 32;
arrstStartupParameter[5].nValue				:= 1;
arrstStartupParameter[6].nRegister			:= 52;
arrstStartupParameter[6].nValue				:= 2;
arrstStartupParameter[7].nRegister			:= 25;
arrstStartupParameter[7].nValue				:= 0;
arrstStartupParameter[8].nRegister			:= 32;
arrstStartupParameter[8].nValue				:= 0;
arrstStartupParameter[9].nRegister			:= 52;
arrstStartupParameter[9].nValue				:= 0;  *)



;
END_ACTION

END_FUNCTION_BLOCK

// POUs/DIOC/TP10/FB_TP10
FUNCTION_BLOCK FB_TP10
VAR_INPUT

	(*Enable bit*)
	bEn					: BOOL:=TRUE; (*enable bit*)

	(*make the TP10 flash green 3 times to know which one you are currently using *)
	bLocate 				: BOOL; (*makes the TP10 flash green 3 times to know which one you are currently using*)

	(*Hardware selection *)
	bRoomAnalyser 		: BOOL; (*FALSE if this instance is a TP10, TRUE if this instance is a Room Analyser*)
	bWallSurface 		: BOOL; (*Not implemented yet*)

	(*led values*)
	arr_bLeds			: ARRAY [0..10] OF BOOL; (*white touch leds (array id 1 is touch button 1)*)
	iIntensityLeds 		: INT := 50; (*intensity of the white leds (0..100)*)

	(*masks of the buttons: true = button disabled*)
	arr_bMasks			: ARRAY [0..10] OF BOOL; (*used to turn off the touch buttons (array id 1 is touch button 1)*)

	(*comment for every button that is visible on the VISU*)
	arr_sButtonComments	: ARRAY [0..10] OF STRING(8); (*comments for every button that is visible on the visualisation*)

	(*Sound level*)
	iHapticIntensity 		: INT := 100; (*intensity of the sound when pressing a button (0..100)*)

	(*sensitivity*)
	iButtonSensitivity 		: DWORD := 0; (*sensitivity of the buttons, only used if value > 0, (values from 1-99 are possible, 99 is the lowest sensitivity, 1 is the highest sensitivity, standard value is 55)*)

	(*RGB values of the TP10: 0-255
	nFillColor := 16#1E8FE03F;
	?1E: intensity in percentage
	?8F: red
	?E0: green
	?3F: blue*)
	dwRgb 				: DWORD;	(*color of the rgb leds*)
	iRGBIntensity			: INT := -1;		(* if intensity > -1 then use this value *)

	(*retrieval times of all sensors*)
	iIntervalRoomtemp	: INT := 3; (*retrieval time of the temperature sensor ( in seconds)*)
	iIntervalRoomHumidity	: INT := 11; (*retrieval time of the humidity sensor ( in seconds)*)
	iIntervalCO2			: INT := 8; (*retrieval time of the CO2 sensor ( in seconds)*)
	iIntervalCO			: INT := 7; (*retrieval time of the CO sensor ( in seconds)*)
	iIntervalVOC			: INT := 5; (*retrieval time of the VOC sensor ( in seconds)*)
	iIntervalIllumination	: INT := 13; (*retrieval time of the Illumination sensor ( in seconds)*)

	(*bool value to reset the TP10*)
	bReset				: BOOL := TRUE; (*true on startup to ensure the device is completely reset when the program is restarted to quickly after the device has been disabled*)
	bResetVOC			: BOOL := FALSE; (*if this input is true, the VOC/eCO2 sensor will be turned off for 1000 cycles*)

END_VAR
VAR_OUTPUT

	(*values of the buttons *)
	qarr_bButtons: ARRAY [0..12] OF BOOL; (*True if a button is pressed (array id 1 is button 1)*)

	(*measurement values *)
	qfRoomTemperature:REAL; (*measurement value of the temperature*)
	qfVOC: REAL;(*measurement value of the VOC*)
	qfCO2:REAL;(*measurement value of the CO2*)
	qfHumidity:REAL;(*measurement value of the humidity*)
	qfLux:REAL;(*measurement value of the lux*)
	qfDewpoint:REAL;(*calculated dewpoint value, dependant on temperature and humidity measurements*)

	(*Analyse data*)
	qdtVersionHw: DATE; (*Hardware version of the dioc device*)
	qdtVersionSw: DATE; (*software version of the dioc device*)
	qdtVersionReg: DATE; (*register version of the dioc device*)
	qsUniqueId: STRING; (*Unique id the dioc device*)
	qrVoltageLevelA: REAL; (*Voltage level on the DIOC-A line*)
	qrVoltageLevelB: REAL; (*Voltage level on the DIOC-B line*)
	qbDeviceActive: BOOL; (*True if the device is active*)

END_VAR
VAR
(* TC3 attribute, will be ignored by TC2 *)
{attribute 'hide_all_locals'}
(* TC2 attribute, will be ignored by TC3 *)
{library private}
(* buttons that can be utilised in the visualisation*)
	_arr_bVisuButtons: ARRAY [0..10] OF BOOL;

(* reset vars *)
	_iReset_Counter:INT;
	_iReset_CounterVOC: INT;

(* startup vars *)
	_RtrigCalibration:R_TRIG;
	_FtrigCalibration:F_TRIG;
	_iLostCalibration:INT;
	_iStateInit:INT;
	_iStateInit_Counter:INT;
	_iStartupListNumber: INT := 1;
	_firstCycle: BOOL := TRUE;
	_iLoadbalance : INT;
	_sLastError : STRING;
	_iCurrentError : UINT;
	_iErrorResetTries : INT;

(* visualisation vars*)
	_iVis: INT;
	_dwVisColor : DWORD;
	_bSelected : BOOL;
	_bPrevVisu : BOOL;
	_bNextVisu :BOOL;
	_RtrigAnalyse :R_TRIG;
	_iLocateCounter : INT;
	_bAnalyse	:BOOL;
	_arrbyRgb	: ARRAY[0..3] OF BYTE;
	_iRgbIntensity : INT;
	(*_byRgbRed : BYTE;
	_byRgbGreen: BYTE;
	_byRgbBlue: BYTE;*)

	(*start*)
	_bInit : BOOL := FALSE;

	(*the communication function block *)
	FB_DIOC_COMM : FB_TP10_COMM;

	(*dewpoint calculation*)
	_iLoadbalanceDewpoint : INT; (*loadbalance to calculate dewpoint*)
END_VAR

(*Wait 0.5s to start the next DIOC device, charging too many DIOC devices at once will give too much current*)
IF NOT _bInit THEN
    DIOC_tonLastStart(IN:=TRUE , PT:= T#500ms);
    IF  NOT DIOC_tonLastStart.Q THEN
    	RETURN;
    END_IF
    DIOC_tonLastStart(IN:=FALSE , PT:= T#500ms); (*resets the timer*)
    _bInit := TRUE;
END_IF

(* falling and rising edge TP10 calibration*)
_RtrigCalibration(CLK:= FB_DIOC_COMM.out.DIOC_TP10.bCalibrationFinished, Q=> );
_FtrigCalibration(CLK:= FB_DIOC_COMM.out.DIOC_TP10.bCalibrationFinished, Q=> );

(* enable reset the device when calibration is lost for 30 cycles. *)
IF _FtrigCalibration.Q THEN
	_iLostCalibration := 1;
END_IF;

IF _iLostCalibration = 30 THEN
	bReset := TRUE;
END_IF;

IF _iLostCalibration < 30 AND _iLostCalibration > 0 AND NOT FB_DIOC_COMM.out.DIOC_TP10.bCalibrationFinished THEN
	_iLostCalibration := _iLostCalibration + 1;
ELSE
	_iLostCalibration := 0;
END_IF

(* reset the device when breset is high, cut off power to device for 1000 cycles to make sure the device has lost all power*)
IF breset OR DIOC_bRestart OR NOT bEn THEN
	_iReset_Counter := 0;
	FB_DIOC_COMM.in.bEnable := FALSE;
	breset := FALSE;
END_IF

IF _iReset_Counter < 1000 THEN
	IF _iReset_Counter = 999 THEN
	    _bInit := FALSE;
	END_IF
	_iReset_Counter := _iReset_Counter +1;
	_iStateInit := 0;
ELSE
	FB_DIOC_COMM.in.bEnable := bEn;
END_IF

(* send startuplist, send all values that need to be sent at startup + set automatic response types of certain measurements,
with synchronisations added in between the messages to not disrupt the flow of the startparameters *)

IF _firstCycle THEN
	StartupList();
END_IF

(* request all static info when the device has been active for some time *)
stateinit();

(* call communication block *)
FB_DIOC_COMM(in:= , out=> , nError=> );

(*save all outputs coming from the tp10*)
(*qarr_bButtons[0]:= dummy*)
qarr_bButtons[1]:=_arr_bVisuButtons[1]  OR FB_DIOC_COMM.out.DIOC_TP10.bR50_TouchButton01;
qarr_bButtons[2]:=_arr_bVisuButtons[2]  OR FB_DIOC_COMM.out.DIOC_TP10.bR50_TouchButton02;
qarr_bButtons[3]:=_arr_bVisuButtons[3]  OR FB_DIOC_COMM.out.DIOC_TP10.bR50_TouchButton03;
qarr_bButtons[4]:=_arr_bVisuButtons[4]  OR FB_DIOC_COMM.out.DIOC_TP10.bR50_TouchButton04;
qarr_bButtons[5]:=_arr_bVisuButtons[5]  OR FB_DIOC_COMM.out.DIOC_TP10.bR50_TouchButton05;
qarr_bButtons[6]:=_arr_bVisuButtons[6]  OR FB_DIOC_COMM.out.DIOC_TP10.bR50_TouchButton06;
qarr_bButtons[7]:=_arr_bVisuButtons[7]  OR FB_DIOC_COMM.out.DIOC_TP10.bR50_TouchButton07;
qarr_bButtons[8]:=_arr_bVisuButtons[8]  OR FB_DIOC_COMM.out.DIOC_TP10.bR50_TouchButton08;
qarr_bButtons[9]:=_arr_bVisuButtons[9]  OR FB_DIOC_COMM.out.DIOC_TP10.bR50_TouchButton09;
qarr_bButtons[10]:=_arr_bVisuButtons[10] OR FB_DIOC_COMM.out.DIOC_TP10.bR50_TouchButton10;

(*enable or disable masks, all masks but the tenth one is enabled when bRoomAnalyser is enabled *)
FB_DIOC_COMM.in.DIOC_TP10.nR52_TouchLedMask := 0;
FB_DIOC_COMM.in.DIOC_TP10.nR52_TouchLedMask.0:= NOT SEL(bRoomAnalyser,arr_bMasks[1],TRUE);
FB_DIOC_COMM.in.DIOC_TP10.nR52_TouchLedMask.1:= NOT SEL(bRoomAnalyser,arr_bMasks[2],TRUE);
FB_DIOC_COMM.in.DIOC_TP10.nR52_TouchLedMask.2:= NOT SEL(bRoomAnalyser,arr_bMasks[3],TRUE);
FB_DIOC_COMM.in.DIOC_TP10.nR52_TouchLedMask.3:= NOT SEL(bRoomAnalyser,arr_bMasks[4],TRUE);
FB_DIOC_COMM.in.DIOC_TP10.nR52_TouchLedMask.4:= NOT SEL(bRoomAnalyser,arr_bMasks[5],TRUE);
FB_DIOC_COMM.in.DIOC_TP10.nR52_TouchLedMask.5:= NOT SEL(bRoomAnalyser,arr_bMasks[6],TRUE);
FB_DIOC_COMM.in.DIOC_TP10.nR52_TouchLedMask.6:= NOT SEL(bRoomAnalyser,arr_bMasks[7],TRUE);
FB_DIOC_COMM.in.DIOC_TP10.nR52_TouchLedMask.7:= NOT SEL(bRoomAnalyser,arr_bMasks[8],TRUE);
FB_DIOC_COMM.in.DIOC_TP10.nR52_TouchLedMask.8:= NOT SEL(bRoomAnalyser,arr_bMasks[9],TRUE);
FB_DIOC_COMM.in.DIOC_TP10.nR52_TouchLedMask.9:= NOT SEL(bRoomAnalyser,arr_bMasks[10],FALSE);(* the button near the fixsus logo can be used to identify the device*)

(*write sensitivity to the TP10*)
IF (iButtonSensitivity > 0) THEN
	FB_DIOC_COMM.in.DIOC_TP10.NR83_ButtonSensitivity :=iButtonSensitivity;
END_IF

IF (NOT bRoomAnalyser) THEN (* only use leds when the device is a TP10, not a multisensor*)
	(*send LED values*)
	FB_DIOC_COMM.in.DIOC_TP10.nR51_TouchLedStatus.0 := arr_bLeds[1];
	FB_DIOC_COMM.in.DIOC_TP10.nR51_TouchLedStatus.1 := arr_bLeds[2];
	FB_DIOC_COMM.in.DIOC_TP10.nR51_TouchLedStatus.2 := arr_bLeds[3];
	FB_DIOC_COMM.in.DIOC_TP10.nR51_TouchLedStatus.3 := arr_bLeds[4];
	FB_DIOC_COMM.in.DIOC_TP10.nR51_TouchLedStatus.4 := arr_bLeds[5];
	FB_DIOC_COMM.in.DIOC_TP10.nR51_TouchLedStatus.5 := arr_bLeds[6];
	FB_DIOC_COMM.in.DIOC_TP10.nR51_TouchLedStatus.6 := arr_bLeds[7];
	FB_DIOC_COMM.in.DIOC_TP10.nR51_TouchLedStatus.7 := arr_bLeds[8];
	FB_DIOC_COMM.in.DIOC_TP10.nR51_TouchLedStatus.8 := arr_bLeds[9];
	FB_DIOC_COMM.in.DIOC_TP10.nR51_TouchLedStatus.9 := arr_bLeds[10];
END_IF

IF bLocate THEN (* make the TP10 flash green 3 times to know which one you are currently using *)
	_iLocateCounter := _iLocateCounter +1;

	FB_DIOC_COMM.in.DIOC_TP10.nR61_RGB_RED := 0 ;
	FB_DIOC_COMM.in.DIOC_TP10.nR61_RGB_BlUE := 0 ;
 	IF ((_iLocateCounter < 100) OR ((_iLocateCounter > 200) AND (_iLocateCounter < 300)) OR (_iLocateCounter > 400)) THEN
		FB_DIOC_COMM.in.DIOC_TP10.nR61_RGB_GREEN := 255 ;
	ELSE
		FB_DIOC_COMM.in.DIOC_TP10.nR61_RGB_GREEN := 0;
	END_IF

	IF _iLocateCounter > 500 THEN
		_iLocateCounter := 0;
		bLocate := FALSE;
	END_IF
ELSE
	IF bRoomAnalyser THEN
		FB_DIOC_COMM.in.DIOC_TP10.nR61_RGB_RED := 0 ;
		FB_DIOC_COMM.in.DIOC_TP10.nR61_RGB_BlUE := 0 ;
		IF qarr_bButtons[10] THEN(* the button near the fixsus logo can be used to identify the device*)
			FB_DIOC_COMM.in.DIOC_TP10.nR61_RGB_GREEN := 255;
		ELSE
			FB_DIOC_COMM.in.DIOC_TP10.nR61_RGB_GREEN := 0;
		END_IF
	ELSE
	(*send RGB LED values*)
	MEMCPY(ADR(_arrbyRgb), ADR(dwRgb), 4);
	IF iRGBIntensity > -1 THEN
		_iRgbIntensity	:= iRGBIntensity;
	ELSE
		_iRgbIntensity	:= BYTE_TO_INT(_arrbyRgb[3]);
	END_IF
	IF _iRgbIntensity > 100 THEN
		_iRgbIntensity := 100;
	ELSIF _iRgbIntensity < 10 THEN
		_iRgbIntensity := 10;
	END_IF

	(* copy requested color to internal variables *)
	FB_DIOC_COMM.in.DIOC_TP10.nR61_RGB_RED := REAL_TO_BYTE(_arrbyRgb[2] * _iRgbIntensity/100.0);
	FB_DIOC_COMM.in.DIOC_TP10.nR61_RGB_GREEN :=  REAL_TO_BYTE(_arrbyRgb[1] * _iRgbIntensity/100.0);
	FB_DIOC_COMM.in.DIOC_TP10.nR61_RGB_BlUE :=  REAL_TO_BYTE(_arrbyRgb[0] * _iRgbIntensity/100.0);

	END_IF
END_IF

(* save measurement values*)
qfRoomTemperature := FB_DIOC_COMM.out.DIOC_TP10.nR21_RoomTemperature;
qfVOC := FB_DIOC_COMM.out.DIOC_TP10.nR27_VOC;
qfCO2 := FB_DIOC_COMM.out.DIOC_TP10.nR25_CO2;
qfHumidity := FB_DIOC_COMM.out.DIOC_TP10.nR23_ROOM_HUMIDITY;
qfLux := (FB_DIOC_COMM.out.DIOC_TP10.nR35_ROOM_ILLUMINATION_LUXL_VALUE + FB_DIOC_COMM.out.DIOC_TP10.nR36_ROOM_ILLUMINATION_LUXH_VALUE*4);

(*reset VOC sensor*)
IF bResetVOC THEN
	bResetVOC := FALSE;
	_iReset_CounterVOC := 1000;
END_IF
IF _iReset_CounterVOC > 1 THEN
	_iReset_CounterVOC := _iReset_CounterVOC - 1;
	(*turn off CO2 first*)
	IF _iReset_CounterVOC = 900 THEN
		FB_DIOC_COMM.in.DIOC_TP10.nR24_CO2_SETUP := 0;
	END_IF
	(*turn off VOC second*)
	IF _iReset_CounterVOC = 800 THEN
		FB_DIOC_COMM.in.DIOC_TP10.nR26_VOC_SETUP := 0;
	END_IF
ELSIF _iReset_CounterVOC = 1 THEN
	_iReset_CounterVOC := _iReset_CounterVOC - 1;
	FB_DIOC_COMM.in.DIOC_TP10.nR24_CO2_SETUP := 1;
	FB_DIOC_COMM.in.DIOC_TP10.nR26_VOC_SETUP := 1;
END_IF

(*loadbalance for dewpoint and temperature offset, only do this every 1100 cycles to save time *)
_iLoadbalanceDewpoint := _iLoadbalanceDewpoint + 1;
IF _iLoadbalanceDewpoint > 1100 THEN
	_iLoadbalanceDewpoint := 0;
	(*calculation of dewpoint in 2 steps*)
	qfDewpoint := LN( (MAX(1,qfHumidity)/100) * EXP( (18.678 - (qfRoomTemperature/234.5)  ) *((qfRoomTemperature) / (257.14 + qfRoomTemperature)) ) );
	qfDewpoint := (257.14 * qfDewpoint) / (18.678 - qfDewpoint) ;
	(*Limit dewpoint to given range*)
	qfDewpoint := LIMIT(0,qfDewpoint,40);
	(*temperature offset for TP10s with fw version between 09/01/2020 and 08/10/2020*)
	IF (qdtVersionSw >= D#2020-01-09) AND (qdtVersionSw < D#2020-02-06) THEN
		FB_DIOC_COMM.in.DIOC_TP10.bR82_Temp_offset := TRUE;
		FB_DIOC_COMM.in.DIOC_TP10.NR82_Temp_offset := 1484;
	ELSIF (qdtVersionSw >= D#2020-02-06) AND (qdtVersionSw < D#2020-10-08) THEN
		FB_DIOC_COMM.in.DIOC_TP10.bR86_Temp_offset := TRUE;
		FB_DIOC_COMM.in.DIOC_TP10.NR86_Temp_offset := 1484;
	END_IF
END_IF

(*loadbalance, only do these tasks every 50 cycles to save time *)
_iLoadbalance := _iLoadbalance + 1;
IF _iLoadbalance > 49 THEN
	_iLoadbalance := 0;

	(* emulation of the TP10s color*)
	_dwVisColor := _arrbyRgb[2] + _arrbyRgb[1] * 256 + _arrbyRgb[0] * 65536;

	(*send haptic intensity *)
	IF iHapticIntensity  > 100 THEN
		iHapticIntensity := 100;
	END_IF
	FB_DIOC_COMM.in.DIOC_TP10.nR57_HapticIntensity := REAL_TO_DWORD((iHapticIntensity * 255) / 100.0);

	(*send led intensity*)
	IF iIntensityLeds  > 100 THEN
		iIntensityLeds := 100;
	END_IF
	FB_DIOC_COMM.in.DIOC_TP10.nR53_LED_Intensity_Max := REAL_TO_DWORD(((100-iIntensityLeds ) * 255) / 100.0);

	(*save static info*)
	qdtVersionHw:=FB_DIOC_COMM.out.DIOC_Gen.dtR04_VersionHW;
	qdtVersionSw:=FB_DIOC_COMM.out.DIOC_Gen.dtR05_VersionSW;
	qdtVersionReg:=FB_DIOC_COMM.out.DIOC_Gen.dtR06_VersionREG;
	qsUniqueId:=FB_DIOC_COMM.out.DIOC_Gen.sR07_UniqueID;

	qrVoltageLevelA:=FB_DIOC_COMM.out.DIOC_Gen.nR09_DiocVoltageA;
	qrVoltageLevelB:=FB_DIOC_COMM.out.DIOC_Gen.nR10_DiocVoltageB;

	qbDeviceActive:=FB_DIOC_COMM.out.DIOC_TP10.bCalibrationFinished;
END_IF


(* Visualisation *)
(*
_RtrigAnalyse(CLK:= _bAnalyse);
IF _RtrigAnalyse.q  AND (CurrentVisu <> DIOC_DEBUGSCHERM) AND DIOC_Debug THEN
	DIOC_DebugLinkPrevScreen:=CurrentVisu;
	CurrentVisu := DIOC_DEBUGSCHERM;
END_IF
IF _bAnalyse AND DIOC_Debug THEN
	DIOC_pDebugged_TP10 := ADRINST();
	_bAnalyse := FALSE;
END_IF*)

IF _bNextVisu THEN
	_iVis := _iVis + 1;
	_bNextVisu := FALSE;
END_IF

IF _bPrevVisu THEN
	_iVis := _iVis - 1;
	_bPrevVisu := FALSE;
END_IF

IF _iVis > 1 THEN
	_iVis := 1;
END_IF;

IF _iVis < 0 THEN
	_iVis := 0;
END_IF;

IF bRoomAnalyser THEN
	_iVis := 1;
END_IF

_firstCycle := FALSE;

ACTION StartupList:
_iStartupListNumber := 1;
(*change transmit offset*)
FB_DIOC_COMM.in.DIOC_TP10.arrstStartupParameter[_iStartupListNumber].nRegister:=DIOC_R84_TRANSMIT_DELAY;
FB_DIOC_COMM.in.DIOC_TP10.arrstStartupParameter[_iStartupListNumber].nValue:=15;

_iStartupListNumber := _iStartupListNumber +1;
FB_DIOC_COMM.in.DIOC_TP10.arrstStartupParameter[_iStartupListNumber].nRegister:=DIOC_R02_REGISTER_INTERVAL;
FB_DIOC_COMM.in.DIOC_TP10.arrstStartupParameter[_iStartupListNumber].nValue:=19;

_iStartupListNumber := _iStartupListNumber +1;
FB_DIOC_COMM.in.DIOC_TP10.arrstStartupParameter[_iStartupListNumber].nRegister:=DIOC_R01_REGISTER_REQUEST;
FB_DIOC_COMM.in.DIOC_TP10.arrstStartupParameter[_iStartupListNumber].nValue:=INT_TO_DWORD(DIOC_R84_TRANSMIT_DELAY);

(*device enabled*)
_iStartupListNumber := _iStartupListNumber +1;
FB_DIOC_COMM.in.DIOC_TP10.arrstStartupParameter[_iStartupListNumber].nRegister:=DIOC_R02_REGISTER_INTERVAL;
FB_DIOC_COMM.in.DIOC_TP10.arrstStartupParameter[_iStartupListNumber].nValue:=15;

_iStartupListNumber := _iStartupListNumber +1;
FB_DIOC_COMM.in.DIOC_TP10.arrstStartupParameter[_iStartupListNumber].nRegister:=DIOC_R01_REGISTER_REQUEST;
FB_DIOC_COMM.in.DIOC_TP10.arrstStartupParameter[_iStartupListNumber].nValue:=INT_TO_DWORD(DIOC_R11_DEVICE_ENABLE);

(*voltage level A*)
_iStartupListNumber := _iStartupListNumber +1;
FB_DIOC_COMM.in.DIOC_TP10.arrstStartupParameter[_iStartupListNumber].nRegister:=DIOC_R02_REGISTER_INTERVAL;
FB_DIOC_COMM.in.DIOC_TP10.arrstStartupParameter[_iStartupListNumber].nValue:=60;

_iStartupListNumber := _iStartupListNumber +1;
FB_DIOC_COMM.in.DIOC_TP10.arrstStartupParameter[_iStartupListNumber].nRegister:=DIOC_R01_REGISTER_REQUEST;
FB_DIOC_COMM.in.DIOC_TP10.arrstStartupParameter[_iStartupListNumber].nValue:=INT_TO_DWORD(DIOC_R09_VOLTAGE_LEVEL_A);

(*voltage level B*)
_iStartupListNumber := _iStartupListNumber +1;
FB_DIOC_COMM.in.DIOC_TP10.arrstStartupParameter[_iStartupListNumber].nRegister:=DIOC_R02_REGISTER_INTERVAL;
FB_DIOC_COMM.in.DIOC_TP10.arrstStartupParameter[_iStartupListNumber].nValue:=61;

_iStartupListNumber := _iStartupListNumber +1;
FB_DIOC_COMM.in.DIOC_TP10.arrstStartupParameter[_iStartupListNumber].nRegister:=DIOC_R01_REGISTER_REQUEST;
FB_DIOC_COMM.in.DIOC_TP10.arrstStartupParameter[_iStartupListNumber].nValue:=INT_TO_DWORD(DIOC_R10_VOLTAGE_LEVEL_B);

(*buttons*)
_iStartupListNumber := _iStartupListNumber +1;
FB_DIOC_COMM.in.DIOC_TP10.arrstStartupParameter[_iStartupListNumber].nRegister:=DIOC_R02_REGISTER_INTERVAL;
FB_DIOC_COMM.in.DIOC_TP10.arrstStartupParameter[_iStartupListNumber].nValue:=0;

_iStartupListNumber := _iStartupListNumber +1;
FB_DIOC_COMM.in.DIOC_TP10.arrstStartupParameter[_iStartupListNumber].nRegister:=DIOC_R01_REGISTER_REQUEST;
FB_DIOC_COMM.in.DIOC_TP10.arrstStartupParameter[_iStartupListNumber].nValue:=INT_TO_DWORD(TP10_R50_TOUCH_BUTTON_STATUS);

(*sync*)
_iStartupListNumber := _iStartupListNumber +1;
FB_DIOC_COMM.in.DIOC_TP10.arrstStartupParameter[_iStartupListNumber].nRegister:=85;
FB_DIOC_COMM.in.DIOC_TP10.arrstStartupParameter[_iStartupListNumber].nValue:=2730;

(*room temperature*)
_iStartupListNumber := _iStartupListNumber +1;
FB_DIOC_COMM.in.DIOC_TP10.arrstStartupParameter[_iStartupListNumber].nRegister:=DIOC_R02_REGISTER_INTERVAL;
FB_DIOC_COMM.in.DIOC_TP10.arrstStartupParameter[_iStartupListNumber].nValue:=INT_TO_DWORD(iIntervalRoomtemp);

_iStartupListNumber := _iStartupListNumber +1;
FB_DIOC_COMM.in.DIOC_TP10.arrstStartupParameter[_iStartupListNumber].nRegister:=DIOC_R01_REGISTER_REQUEST;
FB_DIOC_COMM.in.DIOC_TP10.arrstStartupParameter[_iStartupListNumber].nValue:=INT_TO_DWORD(TP10_R21_ROOMTEMPERATURE);

(*room humidity*)
_iStartupListNumber := _iStartupListNumber +1;
FB_DIOC_COMM.in.DIOC_TP10.arrstStartupParameter[_iStartupListNumber].nRegister:=DIOC_R02_REGISTER_INTERVAL;
FB_DIOC_COMM.in.DIOC_TP10.arrstStartupParameter[_iStartupListNumber].nValue:=INT_TO_DWORD(iIntervalRoomHumidity);

_iStartupListNumber := _iStartupListNumber +1;
FB_DIOC_COMM.in.DIOC_TP10.arrstStartupParameter[_iStartupListNumber].nRegister:=DIOC_R01_REGISTER_REQUEST;
FB_DIOC_COMM.in.DIOC_TP10.arrstStartupParameter[_iStartupListNumber].nValue:=INT_TO_DWORD(TP10_R23_ROOM_HUMIDITY);

(*room CO2*)
_iStartupListNumber := _iStartupListNumber +1;
FB_DIOC_COMM.in.DIOC_TP10.arrstStartupParameter[_iStartupListNumber].nRegister:=DIOC_R02_REGISTER_INTERVAL;
FB_DIOC_COMM.in.DIOC_TP10.arrstStartupParameter[_iStartupListNumber].nValue:=INT_TO_DWORD(iIntervalCO2);

_iStartupListNumber := _iStartupListNumber +1;
FB_DIOC_COMM.in.DIOC_TP10.arrstStartupParameter[_iStartupListNumber].nRegister:=DIOC_R01_REGISTER_REQUEST;
FB_DIOC_COMM.in.DIOC_TP10.arrstStartupParameter[_iStartupListNumber].nValue:=INT_TO_DWORD(TP10_R25_CO2);

(*room CO*)(*
_iStartupListNumber := _iStartupListNumber +1;
FB_DIOC_COMM.in.DIOC_TP10.arrstStartupParameter[_iStartupListNumber].nRegister:=DIOC_R02_REGISTER_INTERVAL;
FB_DIOC_COMM.in.DIOC_TP10.arrstStartupParameter[_iStartupListNumber].nValue:=iIntervalCO;

_iStartupListNumber := _iStartupListNumber +1;
FB_DIOC_COMM.in.DIOC_TP10.arrstStartupParameter[_iStartupListNumber].nRegister:=DIOC_R01_REGISTER_REQUEST;
FB_DIOC_COMM.in.DIOC_TP10.arrstStartupParameter[_iStartupListNumber].nValue:=TP10_R29_CO;
*)

(*sync*)
_iStartupListNumber := _iStartupListNumber +1;
FB_DIOC_COMM.in.DIOC_TP10.arrstStartupParameter[_iStartupListNumber].nRegister:=85;
FB_DIOC_COMM.in.DIOC_TP10.arrstStartupParameter[_iStartupListNumber].nValue:=2730;

(*room VOC*)
_iStartupListNumber := _iStartupListNumber +1;
FB_DIOC_COMM.in.DIOC_TP10.arrstStartupParameter[_iStartupListNumber].nRegister:=DIOC_R02_REGISTER_INTERVAL;
FB_DIOC_COMM.in.DIOC_TP10.arrstStartupParameter[_iStartupListNumber].nValue:=INT_TO_DWORD(iIntervalVOC);

_iStartupListNumber := _iStartupListNumber +1;
FB_DIOC_COMM.in.DIOC_TP10.arrstStartupParameter[_iStartupListNumber].nRegister:=DIOC_R01_REGISTER_REQUEST;
FB_DIOC_COMM.in.DIOC_TP10.arrstStartupParameter[_iStartupListNumber].nValue:=INT_TO_DWORD(TP10_R27_VOC);

(*room illumination*)
_iStartupListNumber := _iStartupListNumber +1;
FB_DIOC_COMM.in.DIOC_TP10.arrstStartupParameter[_iStartupListNumber].nRegister:=DIOC_R02_REGISTER_INTERVAL;
FB_DIOC_COMM.in.DIOC_TP10.arrstStartupParameter[_iStartupListNumber].nValue:=INT_TO_DWORD(iIntervalIllumination);

_iStartupListNumber := _iStartupListNumber +1;
FB_DIOC_COMM.in.DIOC_TP10.arrstStartupParameter[_iStartupListNumber].nRegister:=DIOC_R01_REGISTER_REQUEST;
FB_DIOC_COMM.in.DIOC_TP10.arrstStartupParameter[_iStartupListNumber].nValue:=INT_TO_DWORD(TP10_R36_ROOM_ILLUMINATION_LUXH_VALUE);

(*temperature adjust*)
(*
_iStartupListNumber := _iStartupListNumber +1;
FB_DIOC_COMM.in.DIOC_TP10.arrstStartupParameter[_iStartupListNumber].nRegister:=TP10_R82_TEMP_OFFSET;
FB_DIOC_COMM.in.DIOC_TP10.arrstStartupParameter[_iStartupListNumber].nValue:=22;*)

(*sync*)
_iStartupListNumber := _iStartupListNumber +1;
FB_DIOC_COMM.in.DIOC_TP10.arrstStartupParameter[_iStartupListNumber].nRegister:=85;
FB_DIOC_COMM.in.DIOC_TP10.arrstStartupParameter[_iStartupListNumber].nValue:=2730;
END_ACTION

ACTION Stateinit:
(* Gradually request all static information at startup of the TP10 *)
CASE _iStateInit OF
	0:
		IF _RtrigCalibration.Q  THEN
		(*_iStateInit:=1;*)
		_iStateInit:=1;
		END_IF
	1:
		_iStateInit_Counter:=_iStateInit_Counter+1;
		IF _iStateInit_Counter>4000 THEN
			_iStateInit:=_iStateInit+1;
			_iStateInit_Counter:=0;
		END_IF
	2:
		FB_DIOC_COMM.in.DIOC_Gen.bR04_Request_HW_Version:=TRUE;
		_iStateInit:=_iStateInit+1;
	3:
		_iStateInit_Counter:=_iStateInit_Counter+1;
		IF FB_DIOC_COMM.out.DIOC_Gen.dtR04_VersionHW <> DWORD_TO_DATE(0) THEN
			_iStateInit:=_iStateInit+1;
			_iStateInit_Counter:=0;
		ELSE
			IF _iStateInit_Counter>1000 THEN
				FB_DIOC_COMM.in.DIOC_Gen.bR04_Request_HW_Version:=TRUE;
				_iStateInit_Counter:=0;
			END_IF
		END_IF
	4:
		FB_DIOC_COMM.in.DIOC_Gen.bR05_Request_SW_Version:=TRUE;
		_iStateInit:=_iStateInit+1;
	5:
			_iStateInit_Counter:=_iStateInit_Counter+1;
		IF FB_DIOC_COMM.out.DIOC_Gen.dtR05_VersionSW <> DWORD_TO_DATE(0) THEN
			_iStateInit:=_iStateInit+1;
			_iStateInit_Counter:=0;
		ELSE
			IF _iStateInit_Counter>1000 THEN
				FB_DIOC_COMM.in.DIOC_Gen.bR05_Request_SW_Version:=TRUE;
				_iStateInit_Counter:=0;
			END_IF
		END_IF
	6:
		FB_DIOC_COMM.in.DIOC_Gen.bR06_Request_Register_Version:=TRUE;
		_iStateInit:=_iStateInit+1;
	7:
			_iStateInit_Counter:=_iStateInit_Counter+1;
		IF FB_DIOC_COMM.out.DIOC_Gen.dtR06_VersionREG <> DWORD_TO_DATE(0) THEN
			_iStateInit:=_iStateInit+1;
			_iStateInit_Counter:=0;
		ELSE
			IF _iStateInit_Counter>1000 THEN
				FB_DIOC_COMM.in.DIOC_Gen.bR06_Request_Register_Version:=TRUE;
				_iStateInit_Counter:=0;
			END_IF
		END_IF
	8:
		FB_DIOC_COMM.in.DIOC_Gen.bR07_Request_Unique_ID:=TRUE;
		_iStateInit:=_iStateInit+1;
	9:
		_iStateInit_Counter:=_iStateInit_Counter+1;
		IF FB_DIOC_COMM.out.DIOC_Gen.sR07_UniqueID <> '' THEN
			_iStateInit:=_iStateInit+1;
			_iStateInit_Counter:=0;
		ELSE
			IF _iStateInit_Counter>800 THEN
				FB_DIOC_COMM.in.DIOC_Gen.bR07_Request_Unique_ID:=TRUE;
				_iStateInit_Counter:=0;
			END_IF
		END_IF
	10:
		IF FB_DIOC_COMM.out.DIOC_Gen.sR13_DtLastError <> _sLastError THEN
			_iCurrentError := FB_DIOC_COMM.out.DIOC_Gen.nR13_ErrorRegisterAdress;
			_iStateInit_Counter:=_iStateInit_Counter+1;
			_iStateInit:=_iStateInit+1;
			_iErrorResetTries := 0;
			_sLastError := FB_DIOC_COMM.out.DIOC_Gen.sR13_DtLastError;
		END_IF

	11: (* reset the sensor to off and read if it is reset.*)
		CASE _iCurrentError OF
		20:
			FB_DIOC_COMM.in.DIOC_TP10.nR20_ROOMTEMPERATURE_SETUP := 0;
			FB_DIOC_COMM.in.DIOC_TP10.bR20_Room_Temperature_Setup := TRUE;
			_iStateInit:=_iStateInit+1;
		22:
			FB_DIOC_COMM.in.DIOC_TP10.nR22_ROOM_HUMIDITY_SETUP := 0;
			FB_DIOC_COMM.in.DIOC_TP10.bR22_Room_Humidity_Setup := TRUE;
			_iStateInit:=_iStateInit+1;
		24:
			FB_DIOC_COMM.in.DIOC_TP10.nR24_CO2_SETUP := 0;
			FB_DIOC_COMM.in.DIOC_TP10.bR24_CO2_Setup := TRUE;
			_iStateInit:=_iStateInit+1;
		26:
			FB_DIOC_COMM.in.DIOC_TP10.nR26_VOC_SETUP := 0;
			FB_DIOC_COMM.in.DIOC_TP10.bR26_VOC_Setup := TRUE;
			_iStateInit:=_iStateInit+1;
		34:
			FB_DIOC_COMM.in.DIOC_TP10.nR34_ROOM_ILLUMINATION_SETUP := 0;
			FB_DIOC_COMM.in.DIOC_TP10.bR34_LUX_Setup := TRUE;
			_iStateInit:=_iStateInit+1;
		ELSE
			_iStateInit:=10;
		END_CASE;
	12:
		CASE _iCurrentError OF
		20:
			IF FB_DIOC_COMM.out.DIOC_TP10.nR20_ROOMTEMPERATURE_SETUP = 0 THEN
				FB_DIOC_COMM.in.DIOC_TP10.nR20_ROOMTEMPERATURE_SETUP := 1;
				FB_DIOC_COMM.in.DIOC_TP10.bR20_Room_Temperature_Setup := TRUE;
				_iStateInit:=_iStateInit+1;
			END_IF;
		22:
			IF FB_DIOC_COMM.out.DIOC_TP10.nR22_ROOM_HUMIDITY_SETUP = 0 THEN
				FB_DIOC_COMM.in.DIOC_TP10.nR22_ROOM_HUMIDITY_SETUP := 1;
				FB_DIOC_COMM.in.DIOC_TP10.bR22_Room_Humidity_Setup := TRUE;
				_iStateInit:=_iStateInit+1;
			END_IF;
		24:
			IF FB_DIOC_COMM.out.DIOC_TP10.nR24_CO2_SETUP = 0 THEN
				FB_DIOC_COMM.in.DIOC_TP10.nR24_CO2_SETUP := 1;
				FB_DIOC_COMM.in.DIOC_TP10.bR24_CO2_Setup := TRUE;
				_iStateInit:=_iStateInit+1;
			END_IF;
		26:
			IF FB_DIOC_COMM.out.DIOC_TP10.nR26_VOC_SETUP = 0 THEN
				FB_DIOC_COMM.in.DIOC_TP10.nR26_VOC_SETUP := 1;
				FB_DIOC_COMM.in.DIOC_TP10.bR26_VOC_Setup	 := TRUE;
				_iStateInit:=_iStateInit+1;
			END_IF;
		34:
			IF FB_DIOC_COMM.out.DIOC_TP10.nR34_ROOM_ILLUMINATION_SETUP = 0 THEN
				FB_DIOC_COMM.in.DIOC_TP10.nR34_ROOM_ILLUMINATION_SETUP := 1;
				FB_DIOC_COMM.in.DIOC_TP10.bR34_LUX_Setup := TRUE;
				_iStateInit:=_iStateInit+1;
			END_IF;
		ELSE
			_iStateInit_Counter:= 10;
		END_CASE;
		IF _iStateInit_Counter>800 THEN
			_iStateInit:=11;
			_iStateInit_Counter:=0;
		END_IF
		_iStateInit_Counter:=_iStateInit_Counter+1;
	13:
		CASE _iCurrentError OF
		20:
			IF FB_DIOC_COMM.out.DIOC_TP10.nR20_ROOMTEMPERATURE_SETUP = 1 THEN
				_iStateInit:=10;
			END_IF;
		22:
			IF FB_DIOC_COMM.out.DIOC_TP10.nR22_ROOM_HUMIDITY_SETUP = 1 THEN
				_iStateInit:=10;
			END_IF;
		24:
			IF FB_DIOC_COMM.out.DIOC_TP10.nR24_CO2_SETUP = 1 THEN
				_iStateInit:=10;
			END_IF;
		26:
			IF FB_DIOC_COMM.out.DIOC_TP10.nR26_VOC_SETUP = 1 THEN
				_iStateInit:=10;
			END_IF;
		34:
			IF FB_DIOC_COMM.out.DIOC_TP10.nR34_ROOM_ILLUMINATION_SETUP = 1 OR FB_DIOC_COMM.out.DIOC_TP10.nR34_ROOM_ILLUMINATION_SETUP = 3 THEN
				_iStateInit:=10;
			END_IF;
		ELSE
			_iStateInit_Counter:= 10;
		END_CASE;
		IF _iStateInit_Counter>800 THEN (* retry if the right info has not been received *)
			_iStateInit:=11;
			_iStateInit_Counter:=0;
			_iErrorResetTries := _iErrorResetTries + 1;
		END_IF
		IF _iErrorResetTries = 10 THEN (* after 10 reset tries the tp10 should restart *)
			breset := TRUE;
		END_IF
		_iStateInit_Counter:=_iStateInit_Counter+1;
END_CASE
END_ACTION

END_FUNCTION_BLOCK

